LIN {X 0,Y 467.584,Z 526.238,A -85,B 0,C 180,E1 -7502.759,E2 -7502.759} C_VEL
LIN {X 0,Y 467.555,Z 526.241,A -85,B 0,C 180,E1 -7505.891,E2 -7505.891} C_VEL
LIN {X 0,Y 467.584,Z 526.242,A -85,B 0,C 180,E1 -7509.146,E2 -7509.146} C_VEL
LIN {X 0,Y 467.589,Z 526.235,A -85,B 0,C 180,E1 -7512.568,E2 -7512.568} C_VEL
LIN {X 0,Y 467.573,Z 526.241,A -85,B 0,C 180,E1 -7515.054,E2 -7515.054} C_VEL
LIN {X 0,Y 467.592,Z 526.243,A -85,B 0,C 180,E1 -7517.441,E2 -7517.441} C_VEL
LIN {X 0,Y 467.585,Z 526.237,A -85,B 0,C 180,E1 -7520.856,E2 -7520.856} C_VEL
LIN {X 0,Y 467.563,Z 526.239,A -85,B 0,C 180,E1 -7524.262,E2 -7524.262} C_VEL
LIN {X 0,Y 467.586,Z 526.241,A -85,B 0,C 180,E1 -7527.322,E2 -7527.322} C_VEL
LIN {X 0,Y 467.574,Z 526.237,A -85,B 0,C 180,E1 -7530.668,E2 -7530.668} C_VEL
LIN {X 0,Y 467.62,Z 526.235,A -85,B 0,C 180,E1 -7533.201,E2 -7533.201} C_VEL
LIN {X 0,Y 467.598,Z 526.234,A -85,B 0,C 180,E1 -7536.469,E2 -7536.469} C_VEL
LIN {X 0,Y 467.628,Z 526.237,A -85,B 0,C 180,E1 -7539.778,E2 -7539.778} C_VEL
LIN {X 0,Y 467.604,Z 526.233,A -85,B 0,C 180,E1 -7542.507,E2 -7542.507} C_VEL
LIN {X 0,Y 467.612,Z 526.234,A -85,B 0,C 180,E1 -7545.197,E2 -7545.197} C_VEL
LIN {X 0,Y 467.662,Z 526.232,A -85,B 0,C 180,E1 -7547.855,E2 -7547.855} C_VEL
LIN {X 0,Y 467.686,Z 526.226,A -85,B 0,C 180,E1 -7551.358,E2 -7551.358} C_VEL
LIN {X 0,Y 467.744,Z 526.221,A -85,B 0,C 180,E1 -7553.963,E2 -7553.963} C_VEL
LIN {X 0,Y 467.865,Z 526.204,A -85,B 0,C 180,E1 -7557.418,E2 -7557.418} C_VEL
LIN {X 0,Y 467.889,Z 526.204,A -85,B 0,C 180,E1 -7560,E2 -7560} C_VEL
LIN {X 0,Y 467.866,Z 526.201,A -85,B 0,C 180,E1 -7562.583,E2 -7562.583} C_VEL
LIN {X 0,Y 467.75,Z 526.221,A -85,B 0,C 180,E1 -7566.038,E2 -7566.038} C_VEL
LIN {X 0,Y 467.687,Z 526.223,A -85,B 0,C 180,E1 -7568.643,E2 -7568.643} C_VEL
LIN {X 0,Y 467.662,Z 526.229,A -85,B 0,C 180,E1 -7572.358,E2 -7572.358} C_VEL
LIN {X 0,Y 467.657,Z 526.234,A -85,B 0,C 180,E1 -7575.885,E2 -7575.885} C_VEL
LIN {X 0,Y 467.63,Z 526.231,A -85,B 0,C 180,E1 -7579.308,E2 -7579.308} C_VEL
LIN {X 0,Y 467.542,Z 526.249,A -85,B 0,C 180,E1 -7582.074,E2 -7582.074} C_VEL
LIN {X 0,Y 467.593,Z 526.235,A -85,B 0,C 180,E1 -7584.888,E2 -7584.888} C_VEL
LIN {X 0,Y 467.628,Z 526.234,A -85,B 0,C 180,E1 -7587.769,E2 -7587.769} C_VEL
LIN {X 0,Y 467.575,Z 526.237,A -85,B 0,C 180,E1 -7591.045,E2 -7591.045} C_VEL
LIN {X 0,Y 467.596,Z 526.242,A -85,B 0,C 180,E1 -7594.242,E2 -7594.242} C_VEL
LIN {X 0,Y 467.557,Z 526.239,A -85,B 0,C 180,E1 -7597.186,E2 -7597.186} C_VEL
LIN {X 0,Y 467.579,Z 526.245,A -85,B 0,C 180,E1 -7600.265,E2 -7600.265} C_VEL
LIN {X 0,Y 467.555,Z 526.241,A -85,B 0,C 180,E1 -7603.745,E2 -7603.745} C_VEL
LIN {X 0,Y 467.561,Z 526.247,A -85,B 0,C 180,E1 -7606.255,E2 -7606.255} C_VEL
LIN {X 0,Y 467.585,Z 526.239,A -85,B 0,C 180,E1 -7608.723,E2 -7608.723} C_VEL
LIN {X 0,Y 467.572,Z 526.24,A -85,B 0,C 180,E1 -7611.955,E2 -7611.955} C_VEL
LIN {X 0,Y 467.571,Z 526.238,A -85,B 0,C 180,E1 -7615.167,E2 -7615.167} C_VEL
LIN {X 0,Y 467.59,Z 526.241,A -85,B 0,C 180,E1 -7618.259,E2 -7618.259} C_VEL
LIN {X 0,Y 467.583,Z 526.238,A -85,B 0,C 180,E1 -7621.25,E2 -7621.25} C_VEL
LIN {X 0,Y 467.642,Z 526.251,A -85,B 0,C 180,E1 -7624.2,E2 -7624.2} C_VEL
LIN {X 0,Y 469.788,Z 537.488,A -85,B 0,C 180,E1 -7626.41,E2 -7626.41} C_VEL
LIN {X 0,Y 469.685,Z 545.066,A -85,B 0,C 180,E1 -7627.8,E2 -7627.8} C_VEL
LIN {X 0,Y 468.864,Z 562.445,A -85,B 0,C 180,E1 -7630.92,E2 -7630.92} C_VEL
LIN {X 0,Y 468.38,Z 574.086,A -85,B 0,C 180,E1 -7632.985,E2 -7632.985} C_VEL
LIN {X 0,Y 471.256,Z 592.032,A -85,B 0,C 180,E1 -7633.385,E2 -7633.385} C_VEL
LIN {X 0,Y 470.5,Z 682.57,A -85,B 0,C 180,E1 -7634.818,E2 -7634.818} C_VEL
LIN {X 0,Y 470.126,Z 695.682,A -85,B 0,C 180,E1 -7635.193,E2 -7635.193} C_VEL
LIN {X 0,Y 469.694,Z 707.78,A -85,B 0,C 180,E1 -7635.705,E2 -7635.705} C_VEL
LIN {X 0,Y 469.237,Z 719.207,A -85,B 0,C 180,E1 -7636.354,E2 -7636.354} C_VEL
LIN {X 0,Y 468.71,Z 731,A -85,B 0,C 180,E1 -7637.225,E2 -7637.225} C_VEL
LIN {X 0,Y 468.271,Z 741.513,A -85,B 0,C 180,E1 -7638.199,E2 -7638.199} C_VEL
LIN {X 0,Y 467.801,Z 750.137,A -85,B 0,C 180,E1 -7639.175,E2 -7639.175} C_VEL
LIN {X 0,Y 467.472,Z 758.092,A -85,B 0,C 180,E1 -7640.261,E2 -7640.261} C_VEL
LIN {X 0,Y 467.129,Z 765.864,A -85,B 0,C 180,E1 -7641.564,E2 -7641.564} C_VEL
LIN {X 0,Y 466.861,Z 773.006,A -85,B 0,C 180,E1 -7643.082,E2 -7643.082} C_VEL
LIN {X 0,Y 466.784,Z 777.763,A -85,B 0,C 180,E1 -7644.383,E2 -7644.383} C_VEL
LIN {X 0,Y 466.653,Z 781.394,A -85,B 0,C 180,E1 -7645.68,E2 -7645.68} C_VEL
LIN {X 0,Y 466.691,Z 783.27,A -85,B 0,C 180,E1 -7646.545,E2 -7646.545} C_VEL
LIN {X 0,Y 466.662,Z 784.674,A -85,B 0,C 180,E1 -7647.409,E2 -7647.409} C_VEL
LIN {X 0,Y 466.619,Z 786.281,A -85,B 0,C 180,E1 -7649.136,E2 -7649.136} C_VEL
LIN {X 0,Y 466.598,Z 786.495,A -85,B 0,C 180,E1 -7649.999,E2 -7649.999} C_VEL
LIN {X 0,Y 466.618,Z 786.274,A -85,B 0,C 180,E1 -7650.862,E2 -7650.862} C_VEL
LIN {X 0,Y 466.662,Z 784.653,A -85,B 0,C 180,E1 -7652.588,E2 -7652.588} C_VEL
LIN {X 0,Y 466.691,Z 783.242,A -85,B 0,C 180,E1 -7653.452,E2 -7653.452} C_VEL
LIN {X 0,Y 466.695,Z 780.279,A -85,B 0,C 180,E1 -7654.75,E2 -7654.75} C_VEL
LIN {X 0,Y 466.776,Z 776.271,A -85,B 0,C 180,E1 -7656.049,E2 -7656.049} C_VEL
LIN {X 0,Y 466.951,Z 770.103,A -85,B 0,C 180,E1 -7657.566,E2 -7657.566} C_VEL
LIN {X 0,Y 467.235,Z 763.371,A -85,B 0,C 180,E1 -7658.868,E2 -7658.868} C_VEL
LIN {X 0,Y 467.58,Z 755.016,A -85,B 0,C 180,E1 -7660.171,E2 -7660.171} C_VEL
LIN {X 0,Y 468.025,Z 746.436,A -85,B 0,C 180,E1 -7661.256,E2 -7661.256} C_VEL
LIN {X 0,Y 468.539,Z 736.228,A -85,B 0,C 180,E1 -7662.305,E2 -7662.305} C_VEL
LIN {X 0,Y 469.004,Z 725.64,A -85,B 0,C 180,E1 -7663.186,E2 -7663.186} C_VEL
LIN {X 0,Y 469.445,Z 713.811,A -85,B 0,C 180,E1 -7663.968,E2 -7663.968} C_VEL
LIN {X 0,Y 469.934,Z 701.861,A -85,B 0,C 180,E1 -7664.561,E2 -7664.561} C_VEL
LIN {X 0,Y 470.29,Z 688.979,A -85,B 0,C 180,E1 -7665.02,E2 -7665.02} C_VEL
LIN {X 0,Y 470.579,Z 675.477,A -85,B 0,C 180,E1 -7665.316,E2 -7665.316} C_VEL
LIN {X 0,Y 471.131,Z 591.332,A -85,B 0,C 180,E1 -7666.634,E2 -7666.634} C_VEL
LIN {X 0,Y 468.368,Z 573.742,A -85,B 0,C 180,E1 -7667.03,E2 -7667.03} C_VEL
LIN {X 0,Y 468.993,Z 557.448,A -85,B 0,C 180,E1 -7669.931,E2 -7669.931} C_VEL
LIN {X 0,Y 469.844,Z 541.073,A -85,B 0,C 180,E1 -7672.885,E2 -7672.885} C_VEL
LIN {X 0,Y 469.768,Z 537.298,A -85,B 0,C 180,E1 -7673.589,E2 -7673.589} C_VEL
LIN {X 0,Y 467.64,Z 526.237,A -85,B 0,C 180,E1 -7675.797,E2 -7675.797} C_VEL
LIN {X 0,Y 467.575,Z 526.245,A -85,B 0,C 180,E1 -7678.748,E2 -7678.748} C_VEL
LIN {X 0,Y 467.581,Z 526.244,A -85,B 0,C 180,E1 -7681.738,E2 -7681.738} C_VEL
LIN {X 0,Y 467.563,Z 526.241,A -85,B 0,C 180,E1 -7684.831,E2 -7684.831} C_VEL
LIN {X 0,Y 467.567,Z 526.243,A -85,B 0,C 180,E1 -7688.042,E2 -7688.042} C_VEL
LIN {X 0,Y 467.591,Z 526.239,A -85,B 0,C 180,E1 -7690.261,E2 -7690.261} C_VEL
LIN {X 0,Y 467.581,Z 526.24,A -85,B 0,C 180,E1 -7692.566,E2 -7692.566} C_VEL
LIN {X 0,Y 467.564,Z 526.245,A -85,B 0,C 180,E1 -7695.052,E2 -7695.052} C_VEL
LIN {X 0,Y 467.582,Z 526.243,A -85,B 0,C 180,E1 -7697.439,E2 -7697.439} C_VEL
LIN {X 0,Y 467.608,Z 526.235,A -85,B 0,C 180,E1 -7700.857,E2 -7700.857} C_VEL
LIN {X 0,Y 467.556,Z 526.241,A -85,B 0,C 180,E1 -7704.259,E2 -7704.259} C_VEL
LIN {X 0,Y 467.574,Z 526.243,A -85,B 0,C 180,E1 -7707.32,E2 -7707.32} C_VEL
LIN {X 0,Y 467.569,Z 526.239,A -85,B 0,C 180,E1 -7710.664,E2 -7710.664} C_VEL
LIN {X 0,Y 467.619,Z 526.234,A -85,B 0,C 180,E1 -7713.199,E2 -7713.199} C_VEL
LIN {X 0,Y 467.583,Z 526.233,A -85,B 0,C 180,E1 -7716.467,E2 -7716.467} C_VEL
LIN {X 0,Y 467.614,Z 526.232,A -85,B 0,C 180,E1 -7719.776,E2 -7719.776} C_VEL
LIN {X 0,Y 467.599,Z 526.235,A -85,B 0,C 180,E1 -7722.506,E2 -7722.506} C_VEL
LIN {X 0,Y 467.599,Z 526.236,A -85,B 0,C 180,E1 -7725.196,E2 -7725.196} C_VEL
LIN {X 0,Y 467.672,Z 526.226,A -85,B 0,C 180,E1 -7727.855,E2 -7727.855} C_VEL
LIN {X 0,Y 467.672,Z 526.23,A -85,B 0,C 180,E1 -7731.357,E2 -7731.357} C_VEL
LIN {X 0,Y 467.733,Z 526.22,A -85,B 0,C 180,E1 -7733.962,E2 -7733.962} C_VEL
LIN {X 0,Y 467.85,Z 526.211,A -85,B 0,C 180,E1 -7737.417,E2 -7737.417} C_VEL
LIN {X 0,Y 467.871,Z 526.203,A -85,B 0,C 180,E1 -7740,E2 -7740} C_VEL
LIN {X 0,Y 467.85,Z 526.203,A -85,B 0,C 180,E1 -7742.583,E2 -7742.583} C_VEL
LIN {X 0,Y 467.741,Z 526.219,A -85,B 0,C 180,E1 -7746.037,E2 -7746.037} C_VEL
LIN {X 0,Y 467.671,Z 526.227,A -85,B 0,C 180,E1 -7748.642,E2 -7748.642} C_VEL
LIN {X 0,Y 467.678,Z 526.226,A -85,B 0,C 180,E1 -7752.379,E2 -7752.379} C_VEL
LIN {X 0,Y 467.637,Z 526.235,A -85,B 0,C 180,E1 -7755.885,E2 -7755.885} C_VEL
LIN {X 0,Y 467.612,Z 526.241,A -85,B 0,C 180,E1 -7759.308,E2 -7759.308} C_VEL
LIN {X 0,Y 467.523,Z 526.248,A -85,B 0,C 180,E1 -7762.074,E2 -7762.074} C_VEL
LIN {X 0,Y 467.591,Z 526.241,A -85,B 0,C 180,E1 -7764.887,E2 -7764.887} C_VEL
LIN {X 0,Y 467.628,Z 526.269,A -85,B 0,C 180,E1 -7767.951,E2 -7767.951} C_VEL
LIN {X 0,Y 469.093,Z 534.649,A -85,B 0,C 180,E1 -7769.877,E2 -7769.877} C_VEL
LIN {X 0,Y 468.524,Z 548.568,A -85,B 0,C 180,E1 -7772.861,E2 -7772.861} C_VEL
LIN {X 0,Y 468.485,Z 549.397,A -85,B 0,C 180,E1 -7773.037,E2 -7773.037} C_VEL
LIN {X 0,Y 471.331,Z 564.269,A -85,B 0,C 180,E1 -7773.396,E2 -7773.396} C_VEL
LIN {X 0,Y 470.507,Z 656.723,A -85,B 0,C 180,E1 -7774.868,E2 -7774.868} C_VEL
LIN {X 0,Y 470.226,Z 670.141,A -85,B 0,C 180,E1 -7775.263,E2 -7775.263} C_VEL
LIN {X 0,Y 469.853,Z 681.913,A -85,B 0,C 180,E1 -7775.771,E2 -7775.771} C_VEL
LIN {X 0,Y 469.439,Z 692.978,A -85,B 0,C 180,E1 -7776.407,E2 -7776.407} C_VEL
LIN {X 0,Y 468.925,Z 704.749,A -85,B 0,C 180,E1 -7777.283,E2 -7777.283} C_VEL
LIN {X 0,Y 468.474,Z 714.85,A -85,B 0,C 180,E1 -7778.224,E2 -7778.224} C_VEL
LIN {X 0,Y 468.041,Z 723.751,A -85,B 0,C 180,E1 -7779.237,E2 -7779.237} C_VEL
LIN {X 0,Y 467.686,Z 731.139,A -85,B 0,C 180,E1 -7780.253,E2 -7780.253} C_VEL
LIN {X 0,Y 467.345,Z 738.241,A -85,B 0,C 180,E1 -7781.427,E2 -7781.427} C_VEL
LIN {X 0,Y 467.031,Z 745.32,A -85,B 0,C 180,E1 -7782.897,E2 -7782.897} C_VEL
LIN {X 0,Y 466.844,Z 750.861,A -85,B 0,C 180,E1 -7784.392,E2 -7784.392} C_VEL
LIN {X 0,Y 466.665,Z 754.261,A -85,B 0,C 180,E1 -7785.6,E2 -7785.6} C_VEL
LIN {X 0,Y 466.645,Z 755.815,A -85,B 0,C 180,E1 -7786.295,E2 -7786.295} C_VEL
LIN {X 0,Y 466.541,Z 757.954,A -85,B 0,C 180,E1 -7787.572,E2 -7787.572} C_VEL
LIN {X 0,Y 466.473,Z 759.216,A -85,B 0,C 180,E1 -7788.877,E2 -7788.877} C_VEL
LIN {X 0,Y 466.495,Z 759.567,A -85,B 0,C 180,E1 -7790.204,E2 -7790.204} C_VEL
LIN {X 0,Y 466.545,Z 758.676,A -85,B 0,C 180,E1 -7791.859,E2 -7791.859} C_VEL
LIN {X 0,Y 466.613,Z 756.359,A -85,B 0,C 180,E1 -7793.503,E2 -7793.503} C_VEL
LIN {X 0,Y 466.747,Z 752.589,A -85,B 0,C 180,E1 -7795.099,E2 -7795.099} C_VEL
LIN {X 0,Y 466.765,Z 751.849,A -85,B 0,C 180,E1 -7795.354,E2 -7795.354} C_VEL
LIN {X 0,Y 466.167,Z 749.789,A -85,B 0,C 180,E1 -7796.032,E2 -7796.032} C_VEL
LIN {X 0,Y 463.443,Z 746.027,A -85,B 0,C 180,E1 -7797.115,E2 -7797.115} C_VEL
LIN {X 0,Y 460.774,Z 741.545,A -85,B 0,C 180,E1 -7798.164,E2 -7798.164} C_VEL
LIN {X 0,Y 460.265,Z 738.355,A -85,B 0,C 180,E1 -7798.782,E2 -7798.782} C_VEL
LIN {X 0,Y 460.686,Z 730.288,A -85,B 0,C 180,E1 -7800.115,E2 -7800.115} C_VEL
LIN {X 0,Y 461.126,Z 721.369,A -85,B 0,C 180,E1 -7801.31,E2 -7801.31} C_VEL
LIN {X 0,Y 461.626,Z 711.879,A -85,B 0,C 180,E1 -7802.346,E2 -7802.346} C_VEL
LIN {X 0,Y 462.226,Z 700.526,A -85,B 0,C 180,E1 -7803.333,E2 -7803.333} C_VEL
LIN {X 0,Y 462.71,Z 688.324,A -85,B 0,C 180,E1 -7804.17,E2 -7804.17} C_VEL
LIN {X 0,Y 463.133,Z 676.128,A -85,B 0,C 180,E1 -7804.797,E2 -7804.797} C_VEL
LIN {X 0,Y 463.552,Z 663.091,A -85,B 0,C 180,E1 -7805.271,E2 -7805.271} C_VEL
LIN {X 0,Y 463.735,Z 651.259,A -85,B 0,C 180,E1 -7805.546,E2 -7805.546} C_VEL
LIN {X 0,Y 464.458,Z 564.756,A -85,B 0,C 180,E1 -7806.922,E2 -7806.922} C_VEL
LIN {X 0,Y 461.484,Z 549.204,A -85,B 0,C 180,E1 -7807.298,E2 -7807.298} C_VEL
LIN {X 0,Y 462.003,Z 535.66,A -85,B 0,C 180,E1 -7810.218,E2 -7810.218} C_VEL
LIN {X 0,Y 460.604,Z 527.111,A -85,B 0,C 180,E1 -7812.176,E2 -7812.176} C_VEL
LIN {X 0,Y 460.561,Z 527.119,A -85,B 0,C 180,E1 -7814.966,E2 -7814.966} C_VEL
LIN {X 0,Y 460.604,Z 527.105,A -85,B 0,C 180,E1 -7817.667,E2 -7817.667} C_VEL
LIN {X 0,Y 460.624,Z 527.106,A -85,B 0,C 180,E1 -7821.225,E2 -7821.225} C_VEL
LIN {X 0,Y 460.698,Z 527.093,A -85,B 0,C 180,E1 -7823.871,E2 -7823.871} C_VEL
LIN {X 0,Y 460.823,Z 527.08,A -85,B 0,C 180,E1 -7827.379,E2 -7827.379} C_VEL
LIN {X 0,Y 460.851,Z 527.074,A -85,B 0,C 180,E1 -7830.001,E2 -7830.001} C_VEL
LIN {X 0,Y 460.822,Z 527.082,A -85,B 0,C 180,E1 -7832.624,E2 -7832.624} C_VEL
LIN {X 0,Y 460.699,Z 527.093,A -85,B 0,C 180,E1 -7836.131,E2 -7836.131} C_VEL
LIN {X 0,Y 460.627,Z 527.107,A -85,B 0,C 180,E1 -7838.777,E2 -7838.777} C_VEL
LIN {X 0,Y 460.612,Z 527.105,A -85,B 0,C 180,E1 -7842.446,E2 -7842.446} C_VEL
LIN {X 0,Y 460.599,Z 527.106,A -85,B 0,C 180,E1 -7845.999,E2 -7845.999} C_VEL
LIN {X 0,Y 460.568,Z 527.112,A -85,B 0,C 180,E1 -7849.617,E2 -7849.617} C_VEL
LIN {X 0,Y 460.51,Z 527.117,A -85,B 0,C 180,E1 -7852.43,E2 -7852.43} C_VEL
LIN {X 0,Y 460.568,Z 527.111,A -85,B 0,C 180,E1 -7855.803,E2 -7855.803} C_VEL
LIN {X 0,Y 460.553,Z 527.111,A -85,B 0,C 180,E1 -7858.234,E2 -7858.234} C_VEL
LIN {X 0,Y 460.522,Z 527.123,A -85,B 0,C 180,E1 -7861.284,E2 -7861.284} C_VEL
LIN {X 0,Y 460.533,Z 527.114,A -85,B 0,C 180,E1 -7864.506,E2 -7864.506} C_VEL
LIN {X 0,Y 460.503,Z 527.122,A -85,B 0,C 180,E1 -7867.624,E2 -7867.624} C_VEL
LIN {X 0,Y 460.545,Z 527.112,A -85,B 0,C 180,E1 -7870.271,E2 -7870.271} C_VEL
LIN {X 0,Y 460.512,Z 527.125,A -85,B 0,C 180,E1 -7873.375,E2 -7873.375} C_VEL
LIN {X 0,Y 460.502,Z 527.118,A -85,B 0,C 180,E1 -7876.626,E2 -7876.626} C_VEL
LIN {X 0,Y 460.545,Z 527.117,A -85,B 0,C 180,E1 -7879.732,E2 -7879.732} C_VEL
LIN {X 0,Y 460.503,Z 527.118,A -85,B 0,C 180,E1 -7882.525,E2 -7882.525} C_VEL
LIN {X 0,Y 460.55,Z 527.118,A -85,B 0,C 180,E1 -7885.625,E2 -7885.625} C_VEL
LIN {X 0,Y 460.541,Z 527.113,A -85,B 0,C 180,E1 -7888.745,E2 -7888.745} C_VEL
LIN {X 0,Y 460.586,Z 527.108,A -85,B 0,C 180,E1 -7892.255,E2 -7892.255} C_VEL
LIN {X 0,Y 460.552,Z 527.112,A -85,B 0,C 180,E1 -7894.706,E2 -7894.706} C_VEL
LIN {X 0,Y 460.516,Z 527.124,A -85,B 0,C 180,E1 -7897.572,E2 -7897.572} C_VEL
LIN {X 0,Y 460.573,Z 527.109,A -85,B 0,C 180,E1 -7900.385,E2 -7900.385} C_VEL
LIN {X 0,Y 460.606,Z 527.109,A -85,B 0,C 180,E1 -7904.003,E2 -7904.003} C_VEL
LIN {X 0,Y 460.615,Z 527.112,A -85,B 0,C 180,E1 -7907.666,E2 -7907.666} C_VEL
LIN {X 0,Y 460.633,Z 527.104,A -85,B 0,C 180,E1 -7911.224,E2 -7911.224} C_VEL
LIN {X 0,Y 460.71,Z 527.099,A -85,B 0,C 180,E1 -7913.871,E2 -7913.871} C_VEL
LIN {X 0,Y 460.806,Z 527.083,A -85,B 0,C 180,E1 -7917.378,E2 -7917.378} C_VEL
LIN {X 0,Y 460.859,Z 527.079,A -85,B 0,C 180,E1 -7920,E2 -7920} C_VEL
LIN {X 0,Y 460.806,Z 527.08,A -85,B 0,C 180,E1 -7922.623,E2 -7922.623} C_VEL
LIN {X 0,Y 460.717,Z 527.096,A -85,B 0,C 180,E1 -7926.13,E2 -7926.13} C_VEL
LIN {X 0,Y 460.634,Z 527.101,A -85,B 0,C 180,E1 -7928.776,E2 -7928.776} C_VEL
LIN {X 0,Y 460.621,Z 527.105,A -85,B 0,C 180,E1 -7932.445,E2 -7932.445} C_VEL
LIN {X 0,Y 460.608,Z 527.113,A -85,B 0,C 180,E1 -7935.998,E2 -7935.998} C_VEL
LIN {X 0,Y 460.576,Z 527.112,A -85,B 0,C 180,E1 -7939.616,E2 -7939.616} C_VEL
LIN {X 0,Y 460.518,Z 527.119,A -85,B 0,C 180,E1 -7942.429,E2 -7942.429} C_VEL
LIN {X 0,Y 460.561,Z 527.115,A -85,B 0,C 180,E1 -7945.798,E2 -7945.798} C_VEL
LIN {X 0,Y 460.56,Z 527.117,A -85,B 0,C 180,E1 -7948.233,E2 -7948.233} C_VEL
LIN {X 0,Y 460.528,Z 527.115,A -85,B 0,C 180,E1 -7951.283,E2 -7951.283} C_VEL
LIN {X 0,Y 460.54,Z 527.117,A -85,B 0,C 180,E1 -7954.505,E2 -7954.505} C_VEL
LIN {X 0,Y 460.509,Z 527.118,A -85,B 0,C 180,E1 -7957.623,E2 -7957.623} C_VEL
LIN {X 0,Y 460.543,Z 527.121,A -85,B 0,C 180,E1 -7960.268,E2 -7960.268} C_VEL
LIN {X 0,Y 460.515,Z 527.116,A -85,B 0,C 180,E1 -7963.374,E2 -7963.374} C_VEL
LIN {X 0,Y 460.506,Z 527.121,A -85,B 0,C 180,E1 -7966.624,E2 -7966.624} C_VEL
LIN {X 0,Y 460.549,Z 527.113,A -85,B 0,C 180,E1 -7969.73,E2 -7969.73} C_VEL
LIN {X 0,Y 460.507,Z 527.123,A -85,B 0,C 180,E1 -7972.523,E2 -7972.523} C_VEL
LIN {X 0,Y 460.553,Z 527.112,A -85,B 0,C 180,E1 -7975.623,E2 -7975.623} C_VEL
LIN {X 0,Y 460.544,Z 527.119,A -85,B 0,C 180,E1 -7978.744,E2 -7978.744} C_VEL
LIN {X 0,Y 460.588,Z 527.115,A -85,B 0,C 180,E1 -7982.253,E2 -7982.253} C_VEL
LIN {X 0,Y 460.639,Z 527.249,A -85,B 0,C 180,E1 -7984.009,E2 -7984.009} C_VEL
LIN {X 0,Y 462.957,Z 539.818,A -85,B 0,C 180,E1 -7986.515,E2 -7986.515} C_VEL
LIN {X 0,Y 462.308,Z 553.699,A -85,B 0,C 180,E1 -7989.068,E2 -7989.068} C_VEL
LIN {X 0,Y 461.536,Z 571.352,A -85,B 0,C 180,E1 -7992.268,E2 -7992.268} C_VEL
LIN {X 0,Y 461.423,Z 573.949,A -85,B 0,C 180,E1 -7992.734,E2 -7992.734} C_VEL
LIN {X 0,Y 464.425,Z 593.483,A -85,B 0,C 180,E1 -7993.165,E2 -7993.165} C_VEL
LIN {X 0,Y 463.643,Z 682.087,A -85,B 0,C 180,E1 -7994.588,E2 -7994.588} C_VEL
LIN {X 0,Y 463.232,Z 695.286,A -85,B 0,C 180,E1 -7994.968,E2 -7994.968} C_VEL
LIN {X 0,Y 462.745,Z 708.554,A -85,B 0,C 180,E1 -7995.542,E2 -7995.542} C_VEL
LIN {X 0,Y 462.222,Z 720.503,A -85,B 0,C 180,E1 -7996.255,E2 -7996.255} C_VEL
LIN {X 0,Y 461.726,Z 731.59,A -85,B 0,C 180,E1 -7997.104,E2 -7997.104} C_VEL
LIN {X 0,Y 461.242,Z 742.316,A -85,B 0,C 180,E1 -7998.128,E2 -7998.128} C_VEL
LIN {X 0,Y 460.734,Z 751.598,A -85,B 0,C 180,E1 -7999.229,E2 -7999.229} C_VEL
LIN {X 0,Y 460.291,Z 760.617,A -85,B 0,C 180,E1 -8000.552,E2 -8000.552} C_VEL
LIN {X 0,Y 460.008,Z 767.882,A -85,B 0,C 180,E1 -8001.874,E2 -8001.874} C_VEL
LIN {X 0,Y 459.75,Z 773.966,A -85,B 0,C 180,E1 -8003.272,E2 -8003.272} C_VEL
LIN {X 0,Y 459.662,Z 778.871,A -85,B 0,C 180,E1 -8004.735,E2 -8004.735} C_VEL
LIN {X 0,Y 459.57,Z 781.18,A -85,B 0,C 180,E1 -8005.614,E2 -8005.614} C_VEL
LIN {X 0,Y 459.587,Z 783.059,A -85,B 0,C 180,E1 -8006.492,E2 -8006.492} C_VEL
LIN {X 0,Y 459.585,Z 784.466,A -85,B 0,C 180,E1 -8007.369,E2 -8007.369} C_VEL
LIN {X 0,Y 459.522,Z 786.075,A -85,B 0,C 180,E1 -8009.122,E2 -8009.122} C_VEL
LIN {X 0,Y 459.53,Z 786.291,A -85,B 0,C 180,E1 -8009.999,E2 -8009.999} C_VEL
LIN {X 0,Y 459.522,Z 786.07,A -85,B 0,C 180,E1 -8010.875,E2 -8010.875} C_VEL
LIN {X 0,Y 459.584,Z 784.448,A -85,B 0,C 180,E1 -8012.628,E2 -8012.628} C_VEL
LIN {X 0,Y 459.586,Z 783.035,A -85,B 0,C 180,E1 -8013.506,E2 -8013.506} C_VEL
LIN {X 0,Y 459.623,Z 780.07,A -85,B 0,C 180,E1 -8014.823,E2 -8014.823} C_VEL
LIN {X 0,Y 459.713,Z 775.019,A -85,B 0,C 180,E1 -8016.429,E2 -8016.429} C_VEL
LIN {X 0,Y 459.934,Z 768.867,A -85,B 0,C 180,E1 -8017.903,E2 -8017.903} C_VEL
LIN {X 0,Y 460.232,Z 761.9,A -85,B 0,C 180,E1 -8019.225,E2 -8019.225} C_VEL
LIN {X 0,Y 460.611,Z 753.172,A -85,B 0,C 180,E1 -8020.549,E2 -8020.549} C_VEL
LIN {X 0,Y 461.118,Z 744.231,A -85,B 0,C 180,E1 -8021.649,E2 -8021.649} C_VEL
LIN {X 0,Y 461.596,Z 734.395,A -85,B 0,C 180,E1 -8022.642,E2 -8022.642} C_VEL
LIN {X 0,Y 462.124,Z 723.639,A -85,B 0,C 180,E1 -8023.521,E2 -8023.521} C_VEL
LIN {X 0,Y 462.635,Z 711.554,A -85,B 0,C 180,E1 -8024.29,E2 -8024.29} C_VEL
LIN {X 0,Y 463.135,Z 698.986,A -85,B 0,C 180,E1 -8024.892,E2 -8024.892} C_VEL
LIN {X 0,Y 463.515,Z 686.861,A -85,B 0,C 180,E1 -8025.301,E2 -8025.301} C_VEL
LIN {X 0,Y 463.787,Z 671.695,A -85,B 0,C 180,E1 -8025.602,E2 -8025.602} C_VEL
LIN {X 0,Y 464.316,Z 591.83,A -85,B 0,C 180,E1 -8026.88,E2 -8026.88} C_VEL
LIN {X 0,Y 461.392,Z 573.556,A -85,B 0,C 180,E1 -8027.296,E2 -8027.296} C_VEL
LIN {X 0,Y 462.094,Z 557.28,A -85,B 0,C 180,E1 -8030.242,E2 -8030.242} C_VEL
LIN {X 0,Y 462.944,Z 540.944,A -85,B 0,C 180,E1 -8033.246,E2 -8033.246} C_VEL
LIN {X 0,Y 462.331,Z 535.913,A -85,B 0,C 180,E1 -8034.23,E2 -8034.23} C_VEL
LIN {X 0,Y 460.587,Z 527.115,A -85,B 0,C 180,E1 -8036.06,E2 -8036.06} C_VEL
LIN {X 0,Y 460.553,Z 527.12,A -85,B 0,C 180,E1 -8038.231,E2 -8038.231} C_VEL
LIN {X 0,Y 460.519,Z 527.124,A -85,B 0,C 180,E1 -8041.282,E2 -8041.282} C_VEL
LIN {X 0,Y 460.529,Z 527.117,A -85,B 0,C 180,E1 -8044.504,E2 -8044.504} C_VEL
LIN {X 0,Y 460.526,Z 527.125,A -85,B 0,C 180,E1 -8047.619,E2 -8047.619} C_VEL
LIN {X 0,Y 460.554,Z 527.116,A -85,B 0,C 180,E1 -8050.271,E2 -8050.271} C_VEL
LIN {X 0,Y 460.503,Z 527.128,A -85,B 0,C 180,E1 -8053.373,E2 -8053.373} C_VEL
LIN {X 0,Y 460.493,Z 527.122,A -85,B 0,C 180,E1 -8056.623,E2 -8056.623} C_VEL
LIN {X 0,Y 460.551,Z 527.117,A -85,B 0,C 180,E1 -8059.727,E2 -8059.727} C_VEL
LIN {X 0,Y 460.521,Z 527.115,A -85,B 0,C 180,E1 -8062.518,E2 -8062.518} C_VEL
LIN {X 0,Y 460.541,Z 527.117,A -85,B 0,C 180,E1 -8065.623,E2 -8065.623} C_VEL
LIN {X 0,Y 460.528,Z 527.116,A -85,B 0,C 180,E1 -8068.743,E2 -8068.743} C_VEL
LIN {X 0,Y 460.55,Z 527.115,A -85,B 0,C 180,E1 -8071.766,E2 -8071.766} C_VEL
LIN {X 0,Y 460.55,Z 527.114,A -85,B 0,C 180,E1 -8074.704,E2 -8074.704} C_VEL
LIN {X 0,Y 460.502,Z 527.125,A -85,B 0,C 180,E1 -8077.57,E2 -8077.57} C_VEL
LIN {X 0,Y 460.559,Z 527.107,A -85,B 0,C 180,E1 -8080.384,E2 -8080.384} C_VEL
LIN {X 0,Y 460.555,Z 527.117,A -85,B 0,C 180,E1 -8083.145,E2 -8083.145} C_VEL
LIN {X 0,Y 460.547,Z 527.116,A -85,B 0,C 180,E1 -8085.867,E2 -8085.867} C_VEL
LIN {X 0,Y 460.621,Z 527.101,A -85,B 0,C 180,E1 -8088.559,E2 -8088.559} C_VEL
LIN {X 0,Y 460.684,Z 527.095,A -85,B 0,C 180,E1 -8092.108,E2 -8092.108} C_VEL
LIN {X 0,Y 460.688,Z 527.096,A -85,B 0,C 180,E1 -8094.748,E2 -8094.748} C_VEL
LIN {X 0,Y 460.815,Z 527.088,A -85,B 0,C 180,E1 -8097.377,E2 -8097.377} C_VEL
LIN {X 0,Y 460.842,Z 527.079,A -85,B 0,C 180,E1 -8100,E2 -8100} C_VEL
LIN {X 0,Y 460.815,Z 527.08,A -85,B 0,C 180,E1 -8102.622,E2 -8102.622} C_VEL
LIN {X 0,Y 460.705,Z 527.095,A -85,B 0,C 180,E1 -8106.13,E2 -8106.13} C_VEL
LIN {X 0,Y 460.618,Z 527.107,A -85,B 0,C 180,E1 -8108.776,E2 -8108.776} C_VEL
LIN {X 0,Y 460.621,Z 527.106,A -85,B 0,C 180,E1 -8112.457,E2 -8112.457} C_VEL
LIN {X 0,Y 460.587,Z 527.113,A -85,B 0,C 180,E1 -8115.998,E2 -8115.998} C_VEL
LIN {X 0,Y 460.558,Z 527.117,A -85,B 0,C 180,E1 -8118.902,E2 -8118.902} C_VEL
LIN {X 0,Y 460.503,Z 527.123,A -85,B 0,C 180,E1 -8121.486,E2 -8121.486} C_VEL
LIN {X 0,Y 460.53,Z 527.119,A -85,B 0,C 180,E1 -8124.332,E2 -8124.332} C_VEL
LIN {X 0,Y 460.598,Z 527.115,A -85,B 0,C 180,E1 -8127.727,E2 -8127.727} C_VEL
LIN {X 0,Y 462.016,Z 534.767,A -85,B 0,C 180,E1 -8129.525,E2 -8129.525} C_VEL
LIN {X 0,Y 461.907,Z 542.158,A -85,B 0,C 180,E1 -8131.152,E2 -8131.152} C_VEL
LIN {X 0,Y 461.546,Z 549.686,A -85,B 0,C 180,E1 -8132.777,E2 -8132.777} C_VEL
LIN {X 0,Y 464.587,Z 565.361,A -85,B 0,C 180,E1 -8133.156,E2 -8133.156} C_VEL
LIN {X 0,Y 463.681,Z 656.87,A -85,B 0,C 180,E1 -8134.637,E2 -8134.637} C_VEL
LIN {X 0,Y 463.412,Z 669.859,A -85,B 0,C 180,E1 -8135.023,E2 -8135.023} C_VEL
LIN {X 0,Y 462.989,Z 682.207,A -85,B 0,C 180,E1 -8135.56,E2 -8135.56} C_VEL
LIN {X 0,Y 462.515,Z 694.146,A -85,B 0,C 180,E1 -8136.268,E2 -8136.268} C_VEL
LIN {X 0,Y 462.011,Z 704.688,A -85,B 0,C 180,E1 -8137.067,E2 -8137.067} C_VEL
LIN {X 0,Y 461.503,Z 715.82,A -85,B 0,C 180,E1 -8138.125,E2 -8138.125} C_VEL
LIN {X 0,Y 461.03,Z 724.511,A -85,B 0,C 180,E1 -8139.142,E2 -8139.142} C_VEL
LIN {X 0,Y 460.568,Z 733.341,A -85,B 0,C 180,E1 -8140.417,E2 -8140.417} C_VEL
LIN {X 0,Y 460.15,Z 741.357,A -85,B 0,C 180,E1 -8141.863,E2 -8141.863} C_VEL
LIN {X 0,Y 459.947,Z 746.821,A -85,B 0,C 180,E1 -8143.104,E2 -8143.104} C_VEL
LIN {X 0,Y 459.716,Z 752.229,A -85,B 0,C 180,E1 -8144.686,E2 -8144.686} C_VEL
LIN {X 0,Y 459.561,Z 755.447,A -85,B 0,C 180,E1 -8145.952,E2 -8145.952} C_VEL
LIN {X 0,Y 459.489,Z 757.776,A -85,B 0,C 180,E1 -8147.236,E2 -8147.236} C_VEL
LIN {X 0,Y 459.389,Z 759.427,A -85,B 0,C 180,E1 -8148.867,E2 -8148.867} C_VEL
LIN {X 0,Y 459.413,Z 759.795,A -85,B 0,C 180,E1 -8150.023,E2 -8150.023} C_VEL
LIN {X 0,Y 459.397,Z 759.374,A -85,B 0,C 180,E1 -8151.279,E2 -8151.279} C_VEL
LIN {X 0,Y 459.458,Z 757.939,A -85,B 0,C 180,E1 -8152.693,E2 -8152.693} C_VEL
LIN {X 0,Y 459.62,Z 755.375,A -85,B 0,C 180,E1 -8154.136,E2 -8154.136} C_VEL
LIN {X 0,Y 459.727,Z 751.44,A -85,B 0,C 180,E1 -8155.64,E2 -8155.64} C_VEL
LIN {X 0,Y 459.969,Z 745.914,A -85,B 0,C 180,E1 -8157.177,E2 -8157.177} C_VEL
LIN {X 0,Y 460.251,Z 738.672,A -85,B 0,C 180,E1 -8158.725,E2 -8158.725} C_VEL
LIN {X 0,Y 460.265,Z 738.355,A -85,B 0,C 180,E1 -8158.782,E2 -8158.782} C_VEL
LIN {X 0,Y 459.779,Z 735.039,A -85,B 0,C 180,E1 -8159.384,E2 -8159.384} C_VEL
LIN {X 0,Y 457.246,Z 729.311,A -85,B 0,C 180,E1 -8160.35,E2 -8160.35} C_VEL
LIN {X 0,Y 454.746,Z 723.099,A -85,B 0,C 180,E1 -8161.271,E2 -8161.271} C_VEL
LIN {X 0,Y 454.312,Z 718.898,A -85,B 0,C 180,E1 -8161.793,E2 -8161.793} C_VEL
LIN {X 0,Y 454.824,Z 708.378,A -85,B 0,C 180,E1 -8162.883,E2 -8162.883} C_VEL
LIN {X 0,Y 455.428,Z 697.388,A -85,B 0,C 180,E1 -8163.787,E2 -8163.787} C_VEL
LIN {X 0,Y 455.938,Z 684.607,A -85,B 0,C 180,E1 -8164.603,E2 -8164.603} C_VEL
LIN {X 0,Y 456.414,Z 671.786,A -85,B 0,C 180,E1 -8165.207,E2 -8165.207} C_VEL
LIN {X 0,Y 456.722,Z 658.866,A -85,B 0,C 180,E1 -8165.619,E2 -8165.619} C_VEL
LIN {X 0,Y 456.98,Z 638.88,A -85,B 0,C 180,E1 -8165.981,E2 -8165.981} C_VEL
LIN {X 0,Y 457.704,Z 565.843,A -85,B 0,C 180,E1 -8167.159,E2 -8167.159} C_VEL
LIN {X 0,Y 454.539,Z 549.358,A -85,B 0,C 180,E1 -8167.572,E2 -8167.572} C_VEL
LIN {X 0,Y 455.078,Z 537.586,A -85,B 0,C 180,E1 -8170.139,E2 -8170.139} C_VEL
LIN {X 0,Y 453.686,Z 528.74,A -85,B 0,C 180,E1 -8172.186,E2 -8172.186} C_VEL
LIN {X 0,Y 453.535,Z 527.992,A -85,B 0,C 180,E1 -8172.413,E2 -8172.413} C_VEL
LIN {X 0,Y 453.535,Z 527.994,A -85,B 0,C 180,E1 -8174.728,E2 -8174.728} C_VEL
LIN {X 0,Y 453.558,Z 527.984,A -85,B 0,C 180,E1 -8177.472,E2 -8177.472} C_VEL
LIN {X 0,Y 453.588,Z 527.984,A -85,B 0,C 180,E1 -8181.088,E2 -8181.088} C_VEL
LIN {X 0,Y 453.666,Z 527.969,A -85,B 0,C 180,E1 -8183.776,E2 -8183.776} C_VEL
LIN {X 0,Y 453.763,Z 527.96,A -85,B 0,C 180,E1 -8187.338,E2 -8187.338} C_VEL
LIN {X 0,Y 453.821,Z 527.95,A -85,B 0,C 180,E1 -8190.001,E2 -8190.001} C_VEL
LIN {X 0,Y 453.763,Z 527.962,A -85,B 0,C 180,E1 -8192.664,E2 -8192.664} C_VEL
LIN {X 0,Y 453.667,Z 527.97,A -85,B 0,C 180,E1 -8196.227,E2 -8196.227} C_VEL
LIN {X 0,Y 453.59,Z 527.986,A -85,B 0,C 180,E1 -8198.915,E2 -8198.915} C_VEL
LIN {X 0,Y 453.562,Z 527.984,A -85,B 0,C 180,E1 -8202.53,E2 -8202.53} C_VEL
LIN {X 0,Y 453.543,Z 527.985,A -85,B 0,C 180,E1 -8206.197,E2 -8206.197} C_VEL
LIN {X 0,Y 453.517,Z 527.995,A -85,B 0,C 180,E1 -8209.041,E2 -8209.041} C_VEL
LIN {X 0,Y 453.476,Z 527.994,A -85,B 0,C 180,E1 -8211.837,E2 -8211.837} C_VEL
LIN {X 0,Y 453.513,Z 527.991,A -85,B 0,C 180,E1 -8214.736,E2 -8214.736} C_VEL
LIN {X 0,Y 453.533,Z 527.986,A -85,B 0,C 180,E1 -8217.961,E2 -8217.961} C_VEL
LIN {X 0,Y 453.467,Z 527.999,A -85,B 0,C 180,E1 -8221.526,E2 -8221.526} C_VEL
LIN {X 0,Y 453.488,Z 527.994,A -85,B 0,C 180,E1 -8224.778,E2 -8224.778} C_VEL
LIN {X 0,Y 453.466,Z 527.994,A -85,B 0,C 180,E1 -8228.313,E2 -8228.313} C_VEL
LIN {X 0,Y 453.497,Z 527.991,A -85,B 0,C 180,E1 -8230.61,E2 -8230.61} C_VEL
LIN {X 0,Y 453.466,Z 528.001,A -85,B 0,C 180,E1 -8233.246,E2 -8233.246} C_VEL
LIN {X 0,Y 453.469,Z 527.997,A -85,B 0,C 180,E1 -8235.78,E2 -8235.78} C_VEL
LIN {X 0,Y 453.482,Z 527.993,A -85,B 0,C 180,E1 -8238.21,E2 -8238.21} C_VEL
LIN {X 0,Y 453.498,Z 527.992,A -85,B 0,C 180,E1 -8240.794,E2 -8240.794} C_VEL
LIN {X 0,Y 453.458,Z 527.998,A -85,B 0,C 180,E1 -8243.918,E2 -8243.918} C_VEL
LIN {X 0,Y 453.487,Z 527.995,A -85,B 0,C 180,E1 -8247.152,E2 -8247.152} C_VEL
LIN {X 0,Y 453.479,Z 527.993,A -85,B 0,C 180,E1 -8250.269,E2 -8250.269} C_VEL
LIN {X 0,Y 453.509,Z 527.994,A -85,B 0,C 180,E1 -8253.295,E2 -8253.295} C_VEL
LIN {X 0,Y 453.507,Z 527.99,A -85,B 0,C 180,E1 -8256.24,E2 -8256.24} C_VEL
LIN {X 0,Y 453.488,Z 527.994,A -85,B 0,C 180,E1 -8259.118,E2 -8259.118} C_VEL
LIN {X 0,Y 453.509,Z 527.993,A -85,B 0,C 180,E1 -8261.945,E2 -8261.945} C_VEL
LIN {X 0,Y 453.546,Z 527.984,A -85,B 0,C 180,E1 -8264.727,E2 -8264.727} C_VEL
LIN {X 0,Y 453.565,Z 527.983,A -85,B 0,C 180,E1 -8268.38,E2 -8268.38} C_VEL
LIN {X 0,Y 453.658,Z 527.975,A -85,B 0,C 180,E1 -8271.986,E2 -8271.986} C_VEL
LIN {X 0,Y 453.675,Z 527.968,A -85,B 0,C 180,E1 -8274.667,E2 -8274.667} C_VEL
LIN {X 0,Y 453.75,Z 527.961,A -85,B 0,C 180,E1 -8277.337,E2 -8277.337} C_VEL
LIN {X 0,Y 453.83,Z 527.955,A -85,B 0,C 180,E1 -8280,E2 -8280} C_VEL
LIN {X 0,Y 453.751,Z 527.959,A -85,B 0,C 180,E1 -8282.664,E2 -8282.664} C_VEL
LIN {X 0,Y 453.684,Z 527.971,A -85,B 0,C 180,E1 -8286.226,E2 -8286.226} C_VEL
LIN {X 0,Y 453.598,Z 527.978,A -85,B 0,C 180,E1 -8288.914,E2 -8288.914} C_VEL
LIN {X 0,Y 453.571,Z 527.983,A -85,B 0,C 180,E1 -8292.529,E2 -8292.529} C_VEL
LIN {X 0,Y 453.552,Z 527.989,A -85,B 0,C 180,E1 -8296.196,E2 -8296.196} C_VEL
LIN {X 0,Y 453.525,Z 527.987,A -85,B 0,C 180,E1 -8299.039,E2 -8299.039} C_VEL
LIN {X 0,Y 453.484,Z 527.997,A -85,B 0,C 180,E1 -8301.836,E2 -8301.836} C_VEL
LIN {X 0,Y 453.509,Z 527.99,A -85,B 0,C 180,E1 -8304.735,E2 -8304.735} C_VEL
LIN {X 0,Y 453.54,Z 527.991,A -85,B 0,C 180,E1 -8307.959,E2 -8307.959} C_VEL
LIN {X 0,Y 453.473,Z 527.995,A -85,B 0,C 180,E1 -8311.525,E2 -8311.525} C_VEL
LIN {X 0,Y 453.495,Z 527.992,A -85,B 0,C 180,E1 -8314.777,E2 -8314.777} C_VEL
LIN {X 0,Y 453.468,Z 528.001,A -85,B 0,C 180,E1 -8318.312,E2 -8318.312} C_VEL
LIN {X 0,Y 453.501,Z 527.993,A -85,B 0,C 180,E1 -8320.609,E2 -8320.609} C_VEL
LIN {X 0,Y 453.467,Z 528.002,A -85,B 0,C 180,E1 -8324.221,E2 -8324.221} C_VEL
LIN {X 0,Y 453.47,Z 527.995,A -85,B 0,C 180,E1 -8327.005,E2 -8327.005} C_VEL
LIN {X 0,Y 453.524,Z 527.992,A -85,B 0,C 180,E1 -8330.553,E2 -8330.553} C_VEL
LIN {X 0,Y 453.461,Z 527.997,A -85,B 0,C 180,E1 -8333.917,E2 -8333.917} C_VEL
LIN {X 0,Y 453.49,Z 527.992,A -85,B 0,C 180,E1 -8337.151,E2 -8337.151} C_VEL
LIN {X 0,Y 453.482,Z 527.999,A -85,B 0,C 180,E1 -8340.268,E2 -8340.268} C_VEL
LIN {X 0,Y 453.522,Z 527.991,A -85,B 0,C 180,E1 -8343.294,E2 -8343.294} C_VEL
LIN {X 0,Y 453.585,Z 528.115,A -85,B 0,C 180,E1 -8343.786,E2 -8343.786} C_VEL
LIN {X 0,Y 455.651,Z 538.942,A -85,B 0,C 180,E1 -8345.99,E2 -8345.99} C_VEL
LIN {X 0,Y 456.037,Z 542.138,A -85,B 0,C 180,E1 -8346.618,E2 -8346.618} C_VEL
LIN {X 0,Y 455.175,Z 558.532,A -85,B 0,C 180,E1 -8349.67,E2 -8349.67} C_VEL
LIN {X 0,Y 454.458,Z 573.76,A -85,B 0,C 180,E1 -8352.466,E2 -8352.466} C_VEL
LIN {X 0,Y 457.595,Z 593.953,A -85,B 0,C 180,E1 -8352.922,E2 -8352.922} C_VEL
LIN {X 0,Y 456.787,Z 682.73,A -85,B 0,C 180,E1 -8354.379,E2 -8354.379} C_VEL
LIN {X 0,Y 456.352,Z 695.65,A -85,B 0,C 180,E1 -8354.764,E2 -8354.764} C_VEL
LIN {X 0,Y 455.859,Z 708.213,A -85,B 0,C 180,E1 -8355.319,E2 -8355.319} C_VEL
LIN {X 0,Y 455.301,Z 720.2,A -85,B 0,C 180,E1 -8356.042,E2 -8356.042} C_VEL
LIN {X 0,Y 454.737,Z 732.229,A -85,B 0,C 180,E1 -8356.983,E2 -8356.983} C_VEL
LIN {X 0,Y 454.274,Z 742.05,A -85,B 0,C 180,E1 -8357.943,E2 -8357.943} C_VEL
LIN {X 0,Y 453.703,Z 751.347,A -85,B 0,C 180,E1 -8359.06,E2 -8359.06} C_VEL
LIN {X 0,Y 453.249,Z 760.377,A -85,B 0,C 180,E1 -8360.404,E2 -8360.404} C_VEL
LIN {X 0,Y 452.939,Z 767.65,A -85,B 0,C 180,E1 -8361.747,E2 -8361.747} C_VEL
LIN {X 0,Y 452.725,Z 772.557,A -85,B 0,C 180,E1 -8362.865,E2 -8362.865} C_VEL
LIN {X 0,Y 452.585,Z 777.325,A -85,B 0,C 180,E1 -8364.206,E2 -8364.206} C_VEL
LIN {X 0,Y 452.492,Z 780.967,A -85,B 0,C 180,E1 -8365.545,E2 -8365.545} C_VEL
LIN {X 0,Y 452.483,Z 782.848,A -85,B 0,C 180,E1 -8366.437,E2 -8366.437} C_VEL
LIN {X 0,Y 452.509,Z 784.259,A -85,B 0,C 180,E1 -8367.328,E2 -8367.328} C_VEL
LIN {X 0,Y 452.429,Z 785.87,A -85,B 0,C 180,E1 -8369.109,E2 -8369.109} C_VEL
LIN {X 0,Y 452.434,Z 786.086,A -85,B 0,C 180,E1 -8369.999,E2 -8369.999} C_VEL
LIN {X 0,Y 452.428,Z 785.866,A -85,B 0,C 180,E1 -8370.889,E2 -8370.889} C_VEL
LIN {X 0,Y 452.508,Z 784.242,A -85,B 0,C 180,E1 -8372.669,E2 -8372.669} C_VEL
LIN {X 0,Y 452.483,Z 782.828,A -85,B 0,C 180,E1 -8373.561,E2 -8373.561} C_VEL
LIN {X 0,Y 452.552,Z 779.861,A -85,B 0,C 180,E1 -8374.898,E2 -8374.898} C_VEL
LIN {X 0,Y 452.628,Z 775.224,A -85,B 0,C 180,E1 -8376.415,E2 -8376.415} C_VEL
LIN {X 0,Y 452.869,Z 768.647,A -85,B 0,C 180,E1 -8378.027,E2 -8378.027} C_VEL
LIN {X 0,Y 453.199,Z 761.676,A -85,B 0,C 180,E1 -8379.37,E2 -8379.37} C_VEL
LIN {X 0,Y 453.601,Z 752.946,A -85,B 0,C 180,E1 -8380.714,E2 -8380.714} C_VEL
LIN {X 0,Y 454.157,Z 744.009,A -85,B 0,C 180,E1 -8381.831,E2 -8381.831} C_VEL
LIN {X 0,Y 454.659,Z 733.471,A -85,B 0,C 180,E1 -8382.907,E2 -8382.907} C_VEL
LIN {X 0,Y 455.29,Z 721.855,A -85,B 0,C 180,E1 -8383.842,E2 -8383.842} C_VEL
LIN {X 0,Y 455.827,Z 709.377,A -85,B 0,C 180,E1 -8384.622,E2 -8384.622} C_VEL
LIN {X 0,Y 456.341,Z 696.739,A -85,B 0,C 180,E1 -8385.205,E2 -8385.205} C_VEL
LIN {X 0,Y 456.791,Z 683.374,A -85,B 0,C 180,E1 -8385.618,E2 -8385.618} C_VEL
LIN {X 0,Y 457.122,Z 654.937,A -85,B 0,C 180,E1 -8386.108,E2 -8386.108} C_VEL
LIN {X 0,Y 457.554,Z 592.789,A -85,B 0,C 180,E1 -8387.123,E2 -8387.123} C_VEL
LIN {X 0,Y 454.454,Z 573.234,A -85,B 0,C 180,E1 -8387.596,E2 -8387.596} C_VEL
LIN {X 0,Y 455.187,Z 557.135,A -85,B 0,C 180,E1 -8390.563,E2 -8390.563} C_VEL
LIN {X 0,Y 456.035,Z 542.079,A -85,B 0,C 180,E1 -8393.379,E2 -8393.379} C_VEL
LIN {X 0,Y 455.131,Z 535.792,A -85,B 0,C 180,E1 -8394.639,E2 -8394.639} C_VEL
LIN {X 0,Y 453.533,Z 527.992,A -85,B 0,C 180,E1 -8396.31,E2 -8396.31} C_VEL
LIN {X 0,Y 453.509,Z 527.997,A -85,B 0,C 180,E1 -8398.71,E2 -8398.71} C_VEL
LIN {X 0,Y 453.462,Z 528.002,A -85,B 0,C 180,E1 -8401.798,E2 -8401.798} C_VEL
LIN {X 0,Y 453.477,Z 527.997,A -85,B 0,C 180,E1 -8404.988,E2 -8404.988} C_VEL
LIN {X 0,Y 453.48,Z 527.997,A -85,B 0,C 180,E1 -8408.308,E2 -8408.308} C_VEL
LIN {X 0,Y 453.511,Z 527.993,A -85,B 0,C 180,E1 -8410.605,E2 -8410.605} C_VEL
LIN {X 0,Y 453.467,Z 527.998,A -85,B 0,C 180,E1 -8414.219,E2 -8414.219} C_VEL
LIN {X 0,Y 453.456,Z 528.001,A -85,B 0,C 180,E1 -8417.004,E2 -8417.004} C_VEL
LIN {X 0,Y 453.524,Z 527.988,A -85,B 0,C 180,E1 -8420.553,E2 -8420.553} C_VEL
LIN {X 0,Y 453.45,Z 528,A -85,B 0,C 180,E1 -8423.916,E2 -8423.916} C_VEL
LIN {X 0,Y 453.475,Z 527.997,A -85,B 0,C 180,E1 -8427.15,E2 -8427.15} C_VEL
LIN {X 0,Y 453.505,Z 527.991,A -85,B 0,C 180,E1 -8430.27,E2 -8430.27} C_VEL
LIN {X 0,Y 453.505,Z 527.992,A -85,B 0,C 180,E1 -8433.293,E2 -8433.293} C_VEL
LIN {X 0,Y 453.494,Z 527.988,A -85,B 0,C 180,E1 -8436.238,E2 -8436.238} C_VEL
LIN {X 0,Y 453.473,Z 527.999,A -85,B 0,C 180,E1 -8439.117,E2 -8439.117} C_VEL
LIN {X 0,Y 453.502,Z 527.993,A -85,B 0,C 180,E1 -8441.944,E2 -8441.944} C_VEL
LIN {X 0,Y 453.53,Z 527.984,A -85,B 0,C 180,E1 -8444.726,E2 -8444.726} C_VEL
LIN {X 0,Y 453.591,Z 527.983,A -85,B 0,C 180,E1 -8447.471,E2 -8447.471} C_VEL
LIN {X 0,Y 453.582,Z 527.985,A -85,B 0,C 180,E1 -8451.086,E2 -8451.086} C_VEL
LIN {X 0,Y 453.667,Z 527.974,A -85,B 0,C 180,E1 -8453.774,E2 -8453.774} C_VEL
LIN {X 0,Y 453.756,Z 527.966,A -85,B 0,C 180,E1 -8457.336,E2 -8457.336} C_VEL
LIN {X 0,Y 453.813,Z 527.954,A -85,B 0,C 180,E1 -8460,E2 -8460} C_VEL
LIN {X 0,Y 453.756,Z 527.959,A -85,B 0,C 180,E1 -8462.663,E2 -8462.663} C_VEL
LIN {X 0,Y 453.671,Z 527.971,A -85,B 0,C 180,E1 -8466.225,E2 -8466.225} C_VEL
LIN {X 0,Y 453.582,Z 527.984,A -85,B 0,C 180,E1 -8468.913,E2 -8468.913} C_VEL
LIN {X 0,Y 453.589,Z 527.982,A -85,B 0,C 180,E1 -8472.551,E2 -8472.551} C_VEL
LIN {X 0,Y 453.532,Z 527.991,A -85,B 0,C 180,E1 -8476.196,E2 -8476.196} C_VEL
LIN {X 0,Y 453.508,Z 527.996,A -85,B 0,C 180,E1 -8479.041,E2 -8479.041} C_VEL
LIN {X 0,Y 453.464,Z 528.001,A -85,B 0,C 180,E1 -8481.836,E2 -8481.836} C_VEL
LIN {X 0,Y 453.502,Z 527.996,A -85,B 0,C 180,E1 -8484.735,E2 -8484.735} C_VEL
LIN {X 0,Y 453.571,Z 528.018,A -85,B 0,C 180,E1 -8487.512,E2 -8487.512} C_VEL
LIN {X 0,Y 455.144,Z 536.84,A -85,B 0,C 180,E1 -8489.611,E2 -8489.611} C_VEL
LIN {X 0,Y 454.772,Z 546.69,A -85,B 0,C 180,E1 -8491.795,E2 -8491.795} C_VEL
LIN {X 0,Y 454.655,Z 550.077,A -85,B 0,C 180,E1 -8492.501,E2 -8492.501} C_VEL
LIN {X 0,Y 457.821,Z 566.629,A -85,B 0,C 180,E1 -8492.91,E2 -8492.91} C_VEL
LIN {X 0,Y 456.876,Z 656.761,A -85,B 0,C 180,E1 -8494.392,E2 -8494.392} C_VEL
LIN {X 0,Y 456.555,Z 669.534,A -85,B 0,C 180,E1 -8494.77,E2 -8494.77} C_VEL
LIN {X 0,Y 456.137,Z 682.272,A -85,B 0,C 180,E1 -8495.329,E2 -8495.329} C_VEL
LIN {X 0,Y 455.66,Z 693.707,A -85,B 0,C 180,E1 -8496.007,E2 -8496.007} C_VEL
LIN {X 0,Y 455.072,Z 705.503,A -85,B 0,C 180,E1 -8496.917,E2 -8496.917} C_VEL
LIN {X 0,Y 454.528,Z 716.156,A -85,B 0,C 180,E1 -8497.95,E2 -8497.95} C_VEL
LIN {X 0,Y 454.023,Z 725.238,A -85,B 0,C 180,E1 -8499.04,E2 -8499.04} C_VEL
LIN {X 0,Y 453.541,Z 733.726,A -85,B 0,C 180,E1 -8500.295,E2 -8500.295} C_VEL
LIN {X 0,Y 453.159,Z 740.539,A -85,B 0,C 180,E1 -8501.529,E2 -8501.529} C_VEL
LIN {X 0,Y 452.884,Z 747.299,A -85,B 0,C 180,E1 -8503.063,E2 -8503.063} C_VEL
LIN {X 0,Y 452.661,Z 751.938,A -85,B 0,C 180,E1 -8504.425,E2 -8504.425} C_VEL
LIN {X 0,Y 452.5,Z 755.156,A -85,B 0,C 180,E1 -8505.662,E2 -8505.662} C_VEL
LIN {X 0,Y 452.423,Z 757.508,A -85,B 0,C 180,E1 -8506.894,E2 -8506.894} C_VEL
LIN {X 0,Y 452.319,Z 759.167,A -85,B 0,C 180,E1 -8508.228,E2 -8508.228} C_VEL
LIN {X 0,Y 452.297,Z 759.93,A -85,B 0,C 180,E1 -8509.586,E2 -8509.586} C_VEL
LIN {X 0,Y 452.295,Z 759.752,A -85,B 0,C 180,E1 -8510.979,E2 -8510.979} C_VEL
LIN {X 0,Y 452.365,Z 758.17,A -85,B 0,C 180,E1 -8512.708,E2 -8512.708} C_VEL
LIN {X 0,Y 452.555,Z 755.114,A -85,B 0,C 180,E1 -8514.404,E2 -8514.404} C_VEL
LIN {X 0,Y 452.68,Z 750.687,A -85,B 0,C 180,E1 -8516.021,E2 -8516.021} C_VEL
LIN {X 0,Y 452.911,Z 745.759,A -85,B 0,C 180,E1 -8517.371,E2 -8517.371} C_VEL
LIN {X 0,Y 453.232,Z 738.689,A -85,B 0,C 180,E1 -8518.888,E2 -8518.888} C_VEL
LIN {X 0,Y 453.704,Z 730.343,A -85,B 0,C 180,E1 -8520.287,E2 -8520.287} C_VEL
LIN {X 0,Y 454.162,Z 721.547,A -85,B 0,C 180,E1 -8521.481,E2 -8521.481} C_VEL
LIN {X 0,Y 454.312,Z 718.898,A -85,B 0,C 180,E1 -8521.793,E2 -8521.793} C_VEL
LIN {X 0,Y 453.896,Z 714.565,A -85,B 0,C 180,E1 -8522.291,E2 -8522.291} C_VEL
LIN {X 0,Y 451.498,Z 707.29,A -85,B 0,C 180,E1 -8523.085,E2 -8523.085} C_VEL
LIN {X 0,Y 449.09,Z 699.588,A -85,B 0,C 180,E1 -8523.816,E2 -8523.816} C_VEL
LIN {X 0,Y 448.663,Z 694.498,A -85,B 0,C 180,E1 -8524.211,E2 -8524.211} C_VEL
LIN {X 0,Y 449.176,Z 682.389,A -85,B 0,C 180,E1 -8524.95,E2 -8524.95} C_VEL
LIN {X 0,Y 449.65,Z 669.223,A -85,B 0,C 180,E1 -8525.533,E2 -8525.533} C_VEL
LIN {X 0,Y 449.987,Z 656.112,A -85,B 0,C 180,E1 -8525.921,E2 -8525.921} C_VEL
LIN {X 0,Y 450.929,Z 566.794,A -85,B 0,C 180,E1 -8527.403,E2 -8527.403} C_VEL
LIN {X 0,Y 447.569,Z 549.596,A -85,B 0,C 180,E1 -8527.832,E2 -8527.832} C_VEL
LIN {X 0,Y 448.067,Z 538.04,A -85,B 0,C 180,E1 -8530.394,E2 -8530.394} C_VEL
LIN {X 0,Y 446.51,Z 528.868,A -85,B 0,C 180,E1 -8532.601,E2 -8532.601} C_VEL
LIN {X 0,Y 446.467,Z 528.87,A -85,B 0,C 180,E1 -8535.414,E2 -8535.414} C_VEL
LIN {X 0,Y 446.513,Z 528.862,A -85,B 0,C 180,E1 -8538.194,E2 -8538.194} C_VEL
LIN {X 0,Y 446.596,Z 528.85,A -85,B 0,C 180,E1 -8541.859,E2 -8541.859} C_VEL
LIN {X 0,Y 446.639,Z 528.849,A -85,B 0,C 180,E1 -8544.584,E2 -8544.584} C_VEL
LIN {X 0,Y 446.707,Z 528.839,A -85,B 0,C 180,E1 -8547.296,E2 -8547.296} C_VEL
LIN {X 0,Y 446.791,Z 528.826,A -85,B 0,C 180,E1 -8550.001,E2 -8550.001} C_VEL
LIN {X 0,Y 446.706,Z 528.841,A -85,B 0,C 180,E1 -8552.707,E2 -8552.707} C_VEL
LIN {X 0,Y 446.637,Z 528.846,A -85,B 0,C 180,E1 -8556.325,E2 -8556.325} C_VEL
LIN {X 0,Y 446.536,Z 528.865,A -85,B 0,C 180,E1 -8559.057,E2 -8559.057} C_VEL
LIN {X 0,Y 446.521,Z 528.864,A -85,B 0,C 180,E1 -8562.731,E2 -8562.731} C_VEL
LIN {X 0,Y 446.495,Z 528.863,A -85,B 0,C 180,E1 -8566.229,E2 -8566.229} C_VEL
LIN {X 0,Y 446.468,Z 528.872,A -85,B 0,C 180,E1 -8569.304,E2 -8569.304} C_VEL
LIN {X 0,Y 446.418,Z 528.872,A -85,B 0,C 180,E1 -8572.201,E2 -8572.201} C_VEL
LIN {X 0,Y 446.458,Z 528.876,A -85,B 0,C 180,E1 -8575.153,E2 -8575.153} C_VEL
LIN {X 0,Y 446.485,Z 528.864,A -85,B 0,C 180,E1 -8578.18,E2 -8578.18} C_VEL
LIN {X 0,Y 446.42,Z 528.874,A -85,B 0,C 180,E1 -8581.776,E2 -8581.776} C_VEL
LIN {X 0,Y 446.43,Z 528.871,A -85,B 0,C 180,E1 -8584.524,E2 -8584.524} C_VEL
LIN {X 0,Y 446.417,Z 528.873,A -85,B 0,C 180,E1 -8588.08,E2 -8588.08} C_VEL
LIN {X 0,Y 446.43,Z 528.874,A -85,B 0,C 180,E1 -8590.919,E2 -8590.919} C_VEL
LIN {X 0,Y 446.426,Z 528.874,A -85,B 0,C 180,E1 -8593.844,E2 -8593.844} C_VEL
LIN {X 0,Y 446.402,Z 528.874,A -85,B 0,C 180,E1 -8596.404,E2 -8596.404} C_VEL
LIN {X 0,Y 446.43,Z 528.875,A -85,B 0,C 180,E1 -8599.083,E2 -8599.083} C_VEL
LIN {X 0,Y 446.413,Z 528.874,A -85,B 0,C 180,E1 -8602.122,E2 -8602.122} C_VEL
LIN {X 0,Y 446.433,Z 528.879,A -85,B 0,C 180,E1 -8605.478,E2 -8605.478} C_VEL
LIN {X 0,Y 446.42,Z 528.872,A -85,B 0,C 180,E1 -8608.701,E2 -8608.701} C_VEL
LIN {X 0,Y 446.489,Z 528.868,A -85,B 0,C 180,E1 -8611.822,E2 -8611.822} C_VEL
LIN {X 0,Y 446.454,Z 528.868,A -85,B 0,C 180,E1 -8614.848,E2 -8614.848} C_VEL
LIN {X 0,Y 446.453,Z 528.869,A -85,B 0,C 180,E1 -8618.246,E2 -8618.246} C_VEL
LIN {X 0,Y 446.458,Z 528.876,A -85,B 0,C 180,E1 -8621.65,E2 -8621.65} C_VEL
LIN {X 0,Y 446.514,Z 528.861,A -85,B 0,C 180,E1 -8624.48,E2 -8624.48} C_VEL
LIN {X 0,Y 446.523,Z 528.862,A -85,B 0,C 180,E1 -8628.194,E2 -8628.194} C_VEL
LIN {X 0,Y 446.607,Z 528.856,A -85,B 0,C 180,E1 -8631.858,E2 -8631.858} C_VEL
LIN {X 0,Y 446.649,Z 528.844,A -85,B 0,C 180,E1 -8634.583,E2 -8634.583} C_VEL
LIN {X 0,Y 446.671,Z 528.844,A -85,B 0,C 180,E1 -8638.197,E2 -8638.197} C_VEL
LIN {X 0,Y 446.8,Z 528.831,A -85,B 0,C 180,E1 -8640,E2 -8640} C_VEL
LIN {X 0,Y 446.697,Z 528.838,A -85,B 0,C 180,E1 -8642.706,E2 -8642.706} C_VEL
LIN {X 0,Y 446.654,Z 528.846,A -85,B 0,C 180,E1 -8646.324,E2 -8646.324} C_VEL
LIN {X 0,Y 446.544,Z 528.857,A -85,B 0,C 180,E1 -8649.056,E2 -8649.056} C_VEL
LIN {X 0,Y 446.529,Z 528.859,A -85,B 0,C 180,E1 -8652.73,E2 -8652.73} C_VEL
LIN {X 0,Y 446.503,Z 528.867,A -85,B 0,C 180,E1 -8656.228,E2 -8656.228} C_VEL
LIN {X 0,Y 446.476,Z 528.866,A -85,B 0,C 180,E1 -8659.303,E2 -8659.303} C_VEL
LIN {X 0,Y 446.426,Z 528.878,A -85,B 0,C 180,E1 -8662.2,E2 -8662.2} C_VEL
LIN {X 0,Y 446.452,Z 528.868,A -85,B 0,C 180,E1 -8665.153,E2 -8665.153} C_VEL
LIN {X 0,Y 446.493,Z 528.871,A -85,B 0,C 180,E1 -8668.179,E2 -8668.179} C_VEL
LIN {X 0,Y 446.426,Z 528.875,A -85,B 0,C 180,E1 -8671.775,E2 -8671.775} C_VEL
LIN {X 0,Y 446.437,Z 528.874,A -85,B 0,C 180,E1 -8674.523,E2 -8674.523} C_VEL
LIN {X 0,Y 446.421,Z 528.878,A -85,B 0,C 180,E1 -8678.079,E2 -8678.079} C_VEL
LIN {X 0,Y 446.429,Z 528.872,A -85,B 0,C 180,E1 -8680.916,E2 -8680.916} C_VEL
LIN {X 0,Y 446.405,Z 528.877,A -85,B 0,C 180,E1 -8683.846,E2 -8683.846} C_VEL
LIN {X 0,Y 446.406,Z 528.881,A -85,B 0,C 180,E1 -8686.403,E2 -8686.403} C_VEL
LIN {X 0,Y 446.434,Z 528.871,A -85,B 0,C 180,E1 -8689.082,E2 -8689.082} C_VEL
LIN {X 0,Y 446.437,Z 528.873,A -85,B 0,C 180,E1 -8691.918,E2 -8691.918} C_VEL
LIN {X 0,Y 446.436,Z 528.87,A -85,B 0,C 180,E1 -8695.476,E2 -8695.476} C_VEL
LIN {X 0,Y 446.423,Z 528.878,A -85,B 0,C 180,E1 -8698.699,E2 -8698.699} C_VEL
LIN {X 0,Y 446.492,Z 528.867,A -85,B 0,C 180,E1 -8701.821,E2 -8701.821} C_VEL
LIN {X 0,Y 446.533,Z 528.968,A -85,B 0,C 180,E1 -8703.556,E2 -8703.556} C_VEL
LIN {X 0,Y 448.771,Z 540.645,A -85,B 0,C 180,E1 -8705.971,E2 -8705.971} C_VEL
LIN {X 0,Y 449.04,Z 544.446,A -85,B 0,C 180,E1 -8706.721,E2 -8706.721} C_VEL
LIN {X 0,Y 448.084,Z 560.827,A -85,B 0,C 180,E1 -8709.813,E2 -8709.813} C_VEL
LIN {X 0,Y 447.485,Z 573.585,A -85,B 0,C 180,E1 -8712.194,E2 -8712.194} C_VEL
LIN {X 0,Y 450.741,Z 594.297,A -85,B 0,C 180,E1 -8712.672,E2 -8712.672} C_VEL
LIN {X 0,Y 449.912,Z 682.023,A -85,B 0,C 180,E1 -8714.134,E2 -8714.134} C_VEL
LIN {X 0,Y 449.497,Z 695.107,A -85,B 0,C 180,E1 -8714.526,E2 -8714.526} C_VEL
LIN {X 0,Y 449,Z 707.765,A -85,B 0,C 180,E1 -8715.09,E2 -8715.09} C_VEL
LIN {X 0,Y 448.411,Z 719.833,A -85,B 0,C 180,E1 -8715.823,E2 -8715.823} C_VEL
LIN {X 0,Y 447.822,Z 731.325,A -85,B 0,C 180,E1 -8716.727,E2 -8716.727} C_VEL
LIN {X 0,Y 447.295,Z 741.753,A -85,B 0,C 180,E1 -8717.752,E2 -8717.752} C_VEL
LIN {X 0,Y 446.702,Z 751.079,A -85,B 0,C 180,E1 -8718.887,E2 -8718.887} C_VEL
LIN {X 0,Y 446.221,Z 760.127,A -85,B 0,C 180,E1 -8720.251,E2 -8720.251} C_VEL
LIN {X 0,Y 445.866,Z 767.414,A -85,B 0,C 180,E1 -8721.615,E2 -8721.615} C_VEL
LIN {X 0,Y 445.646,Z 772.332,A -85,B 0,C 180,E1 -8722.751,E2 -8722.751} C_VEL
LIN {X 0,Y 445.496,Z 776.511,A -85,B 0,C 180,E1 -8723.925,E2 -8723.925} C_VEL
LIN {X 0,Y 445.418,Z 780.755,A -85,B 0,C 180,E1 -8725.474,E2 -8725.474} C_VEL
LIN {X 0,Y 445.382,Z 782.637,A -85,B 0,C 180,E1 -8726.38,E2 -8726.38} C_VEL
LIN {X 0,Y 445.434,Z 784.052,A -85,B 0,C 180,E1 -8727.286,E2 -8727.286} C_VEL
LIN {X 0,Y 445.339,Z 785.664,A -85,B 0,C 180,E1 -8729.094,E2 -8729.094} C_VEL
LIN {X 0,Y 445.342,Z 785.882,A -85,B 0,C 180,E1 -8729.999,E2 -8729.999} C_VEL
LIN {X 0,Y 445.339,Z 785.662,A -85,B 0,C 180,E1 -8730.903,E2 -8730.903} C_VEL
LIN {X 0,Y 445.433,Z 784.037,A -85,B 0,C 180,E1 -8732.712,E2 -8732.712} C_VEL
LIN {X 0,Y 445.381,Z 782.622,A -85,B 0,C 180,E1 -8733.618,E2 -8733.618} C_VEL
LIN {X 0,Y 445.481,Z 779.655,A -85,B 0,C 180,E1 -8734.976,E2 -8734.976} C_VEL
LIN {X 0,Y 445.576,Z 774.192,A -85,B 0,C 180,E1 -8736.747,E2 -8736.747} C_VEL
LIN {X 0,Y 445.802,Z 768.445,A -85,B 0,C 180,E1 -8738.155,E2 -8738.155} C_VEL
LIN {X 0,Y 446.148,Z 761.477,A -85,B 0,C 180,E1 -8739.519,E2 -8739.519} C_VEL
LIN {X 0,Y 446.589,Z 752.75,A -85,B 0,C 180,E1 -8740.884,E2 -8740.884} C_VEL
LIN {X 0,Y 447.203,Z 743.815,A -85,B 0,C 180,E1 -8742.017,E2 -8742.017} C_VEL
LIN {X 0,Y 447.752,Z 732.921,A -85,B 0,C 180,E1 -8743.143,E2 -8743.143} C_VEL
LIN {X 0,Y 448.371,Z 721.664,A -85,B 0,C 180,E1 -8744.06,E2 -8744.06} C_VEL
LIN {X 0,Y 448.958,Z 709.192,A -85,B 0,C 180,E1 -8744.851,E2 -8744.851} C_VEL
LIN {X 0,Y 449.488,Z 696.573,A -85,B 0,C 180,E1 -8745.442,E2 -8745.442} C_VEL
LIN {X 0,Y 449.967,Z 683.245,A -85,B 0,C 180,E1 -8745.861,E2 -8745.861} C_VEL
LIN {X 0,Y 450.264,Z 656.346,A -85,B 0,C 180,E1 -8746.337,E2 -8746.337} C_VEL
LIN {X 0,Y 450.827,Z 593.889,A -85,B 0,C 180,E1 -8747.37,E2 -8747.37} C_VEL
LIN {X 0,Y 447.522,Z 572.998,A -85,B 0,C 180,E1 -8747.89,E2 -8747.89} C_VEL
LIN {X 0,Y 448.321,Z 557,A -85,B 0,C 180,E1 -8750.892,E2 -8750.892} C_VEL
LIN {X 0,Y 449.098,Z 543.214,A -85,B 0,C 180,E1 -8753.517,E2 -8753.517} C_VEL
LIN {X 0,Y 447.911,Z 535.703,A -85,B 0,C 180,E1 -8755.063,E2 -8755.063} C_VEL
LIN {X 0,Y 446.483,Z 528.87,A -85,B 0,C 180,E1 -8756.549,E2 -8756.549} C_VEL
LIN {X 0,Y 446.447,Z 528.878,A -85,B 0,C 180,E1 -8759.208,E2 -8759.208} C_VEL
LIN {X 0,Y 446.419,Z 528.876,A -85,B 0,C 180,E1 -8762.36,E2 -8762.36} C_VEL
LIN {X 0,Y 446.417,Z 528.88,A -85,B 0,C 180,E1 -8765.624,E2 -8765.624} C_VEL
LIN {X 0,Y 446.47,Z 528.873,A -85,B 0,C 180,E1 -8769.022,E2 -8769.022} C_VEL
LIN {X 0,Y 446.432,Z 528.875,A -85,B 0,C 180,E1 -8772.276,E2 -8772.276} C_VEL
LIN {X 0,Y 446.448,Z 528.875,A -85,B 0,C 180,E1 -8775.102,E2 -8775.102} C_VEL
LIN {X 0,Y 446.428,Z 528.874,A -85,B 0,C 180,E1 -8778.608,E2 -8778.608} C_VEL
LIN {X 0,Y 446.466,Z 528.87,A -85,B 0,C 180,E1 -8780.975,E2 -8780.975} C_VEL
LIN {X 0,Y 446.414,Z 528.875,A -85,B 0,C 180,E1 -8784.373,E2 -8784.373} C_VEL
LIN {X 0,Y 446.415,Z 528.879,A -85,B 0,C 180,E1 -8787.637,E2 -8787.637} C_VEL
LIN {X 0,Y 446.461,Z 528.869,A -85,B 0,C 180,E1 -8790.791,E2 -8790.791} C_VEL
LIN {X 0,Y 446.468,Z 528.871,A -85,B 0,C 180,E1 -8793.847,E2 -8793.847} C_VEL
LIN {X 0,Y 446.419,Z 528.871,A -85,B 0,C 180,E1 -8796.822,E2 -8796.822} C_VEL
LIN {X 0,Y 446.435,Z 528.87,A -85,B 0,C 180,E1 -8799.736,E2 -8799.736} C_VEL
LIN {X 0,Y 446.453,Z 528.87,A -85,B 0,C 180,E1 -8802.596,E2 -8802.596} C_VEL
LIN {X 0,Y 446.461,Z 528.872,A -85,B 0,C 180,E1 -8805.412,E2 -8805.412} C_VEL
LIN {X 0,Y 446.529,Z 528.857,A -85,B 0,C 180,E1 -8808.193,E2 -8808.193} C_VEL
LIN {X 0,Y 446.589,Z 528.853,A -85,B 0,C 180,E1 -8811.857,E2 -8811.857} C_VEL
LIN {X 0,Y 446.636,Z 528.846,A -85,B 0,C 180,E1 -8814.582,E2 -8814.582} C_VEL
LIN {X 0,Y 446.7,Z 528.845,A -85,B 0,C 180,E1 -8817.294,E2 -8817.294} C_VEL
LIN {X 0,Y 446.783,Z 528.83,A -85,B 0,C 180,E1 -8820,E2 -8820} C_VEL
LIN {X 0,Y 446.7,Z 528.838,A -85,B 0,C 180,E1 -8822.705,E2 -8822.705} C_VEL
LIN {X 0,Y 446.64,Z 528.847,A -85,B 0,C 180,E1 -8826.323,E2 -8826.323} C_VEL
LIN {X 0,Y 446.528,Z 528.864,A -85,B 0,C 180,E1 -8829.055,E2 -8829.055} C_VEL
LIN {X 0,Y 446.522,Z 528.863,A -85,B 0,C 180,E1 -8832.729,E2 -8832.729} C_VEL
LIN {X 0,Y 446.477,Z 528.87,A -85,B 0,C 180,E1 -8836.459,E2 -8836.459} C_VEL
LIN {X 0,Y 446.457,Z 528.876,A -85,B 0,C 180,E1 -8839.303,E2 -8839.303} C_VEL
LIN {X 0,Y 446.405,Z 528.878,A -85,B 0,C 180,E1 -8842.2,E2 -8842.2} C_VEL
LIN {X 0,Y 446.446,Z 528.875,A -85,B 0,C 180,E1 -8845.152,E2 -8845.152} C_VEL
LIN {X 0,Y 446.516,Z 528.936,A -85,B 0,C 180,E1 -8847.284,E2 -8847.284} C_VEL
LIN {X 0,Y 448.223,Z 538.497,A -85,B 0,C 180,E1 -8849.597,E2 -8849.597} C_VEL
LIN {X 0,Y 447.687,Z 550.091,A -85,B 0,C 180,E1 -8852.202,E2 -8852.202} C_VEL
LIN {X 0,Y 451.078,Z 567.137,A -85,B 0,C 180,E1 -8852.644,E2 -8852.644} C_VEL
LIN {X 0,Y 450.053,Z 656.96,A -85,B 0,C 180,E1 -8854.145,E2 -8854.145} C_VEL
LIN {X 0,Y 449.73,Z 669.971,A -85,B 0,C 180,E1 -8854.539,E2 -8854.539} C_VEL
LIN {X 0,Y 449.3,Z 682.302,A -85,B 0,C 180,E1 -8855.088,E2 -8855.088} C_VEL
LIN {X 0,Y 448.798,Z 693.827,A -85,B 0,C 180,E1 -8855.78,E2 -8855.78} C_VEL
LIN {X 0,Y 448.184,Z 705.789,A -85,B 0,C 180,E1 -8856.716,E2 -8856.716} C_VEL
LIN {X 0,Y 447.562,Z 716.427,A -85,B 0,C 180,E1 -8857.763,E2 -8857.763} C_VEL
LIN {X 0,Y 447,Z 726.2,A -85,B 0,C 180,E1 -8858.969,E2 -8858.969} C_VEL
LIN {X 0,Y 446.472,Z 735.289,A -85,B 0,C 180,E1 -8860.365,E2 -8860.365} C_VEL
LIN {X 0,Y 446.02,Z 742.795,A -85,B 0,C 180,E1 -8861.818,E2 -8861.818} C_VEL
LIN {X 0,Y 445.809,Z 748.021,A -85,B 0,C 180,E1 -8863.086,E2 -8863.086} C_VEL
LIN {X 0,Y 445.512,Z 753.37,A -85,B 0,C 180,E1 -8864.777,E2 -8864.777} C_VEL
LIN {X 0,Y 445.362,Z 757.242,A -85,B 0,C 180,E1 -8866.543,E2 -8866.543} C_VEL
LIN {X 0,Y 445.261,Z 759.102,A -85,B 0,C 180,E1 -8867.888,E2 -8867.888} C_VEL
LIN {X 0,Y 445.199,Z 760.151,A -85,B 0,C 180,E1 -8869.669,E2 -8869.669} C_VEL
LIN {X 0,Y 445.221,Z 760.032,A -85,B 0,C 180,E1 -8870.847,E2 -8870.847} C_VEL
LIN {X 0,Y 445.253,Z 759.129,A -85,B 0,C 180,E1 -8872.111,E2 -8872.111} C_VEL
LIN {X 0,Y 445.349,Z 757.073,A -85,B 0,C 180,E1 -8873.592,E2 -8873.592} C_VEL
LIN {X 0,Y 445.495,Z 753.758,A -85,B 0,C 180,E1 -8875.118,E2 -8875.118} C_VEL
LIN {X 0,Y 445.711,Z 748.948,A -85,B 0,C 180,E1 -8876.689,E2 -8876.689} C_VEL
LIN {X 0,Y 445.949,Z 743.802,A -85,B 0,C 180,E1 -8877.989,E2 -8877.989} C_VEL
LIN {X 0,Y 446.352,Z 736.352,A -85,B 0,C 180,E1 -8879.485,E2 -8879.485} C_VEL
LIN {X 0,Y 446.821,Z 727.979,A -85,B 0,C 180,E1 -8880.819,E2 -8880.819} C_VEL
LIN {X 0,Y 447.35,Z 718.724,A -85,B 0,C 180,E1 -8882.01,E2 -8882.01} C_VEL
LIN {X 0,Y 447.875,Z 708.712,A -85,B 0,C 180,E1 -8883.059,E2 -8883.059} C_VEL
LIN {X 0,Y 448.504,Z 697.765,A -85,B 0,C 180,E1 -8883.977,E2 -8883.977} C_VEL
LIN {X 0,Y 448.663,Z 694.498,A -85,B 0,C 180,E1 -8884.211,E2 -8884.211} C_VEL
LIN {X 0,Y 448.214,Z 689.348,A -85,B 0,C 180,E1 -8884.582,E2 -8884.582} C_VEL
LIN {X 0,Y 445.725,Z 680.858,A -85,B 0,C 180,E1 -8885.167,E2 -8885.167} C_VEL
LIN {X 0,Y 443.272,Z 672.054,A -85,B 0,C 180,E1 -8885.657,E2 -8885.657} C_VEL
LIN {X 0,Y 442.863,Z 666.425,A -85,B 0,C 180,E1 -8885.875,E2 -8885.875} C_VEL
LIN {X 0,Y 443.185,Z 652.917,A -85,B 0,C 180,E1 -8886.227,E2 -8886.227} C_VEL
LIN {X 0,Y 444.113,Z 567.644,A -85,B 0,C 180,E1 -8887.656,E2 -8887.656} C_VEL
LIN {X 0,Y 440.644,Z 549.774,A -85,B 0,C 180,E1 -8888.112,E2 -8888.112} C_VEL
LIN {X 0,Y 441.105,Z 539.359,A -85,B 0,C 180,E1 -8890.454,E2 -8890.454} C_VEL
LIN {X 0,Y 439.462,Z 529.747,A -85,B 0,C 180,E1 -8892.793,E2 -8892.793} C_VEL
LIN {X 0,Y 439.429,Z 529.747,A -85,B 0,C 180,E1 -8896.121,E2 -8896.121} C_VEL
LIN {X 0,Y 439.433,Z 529.749,A -85,B 0,C 180,E1 -8898.937,E2 -8898.937} C_VEL
LIN {X 0,Y 439.595,Z 529.725,A -85,B 0,C 180,E1 -8902.398,E2 -8902.398} C_VEL
LIN {X 0,Y 439.614,Z 529.723,A -85,B 0,C 180,E1 -8904.497,E2 -8904.497} C_VEL
LIN {X 0,Y 439.633,Z 529.718,A -85,B 0,C 180,E1 -8908.169,E2 -8908.169} C_VEL
LIN {X 0,Y 439.761,Z 529.702,A -85,B 0,C 180,E1 -8910.001,E2 -8910.001} C_VEL
LIN {X 0,Y 439.653,Z 529.721,A -85,B 0,C 180,E1 -8912.75,E2 -8912.75} C_VEL
LIN {X 0,Y 439.609,Z 529.722,A -85,B 0,C 180,E1 -8916.427,E2 -8916.427} C_VEL
LIN {X 0,Y 439.498,Z 529.74,A -85,B 0,C 180,E1 -8919.203,E2 -8919.203} C_VEL
LIN {X 0,Y 439.465,Z 529.745,A -85,B 0,C 180,E1 -8922.939,E2 -8922.939} C_VEL
LIN {X 0,Y 439.446,Z 529.741,A -85,B 0,C 180,E1 -8926.35,E2 -8926.35} C_VEL
LIN {X 0,Y 439.402,Z 529.748,A -85,B 0,C 180,E1 -8929.628,E2 -8929.628} C_VEL
LIN {X 0,Y 439.365,Z 529.753,A -85,B 0,C 180,E1 -8932.577,E2 -8932.577} C_VEL
LIN {X 0,Y 439.405,Z 529.749,A -85,B 0,C 180,E1 -8935.586,E2 -8935.586} C_VEL
LIN {X 0,Y 439.418,Z 529.746,A -85,B 0,C 180,E1 -8938.675,E2 -8938.675} C_VEL
LIN {X 0,Y 439.371,Z 529.751,A -85,B 0,C 180,E1 -8942.032,E2 -8942.032} C_VEL
LIN {X 0,Y 439.396,Z 529.755,A -85,B 0,C 180,E1 -8945.341,E2 -8945.341} C_VEL
LIN {X 0,Y 439.385,Z 529.749,A -85,B 0,C 180,E1 -8948.596,E2 -8948.596} C_VEL
LIN {X 0,Y 439.392,Z 529.755,A -85,B 0,C 180,E1 -8951.258,E2 -8951.258} C_VEL
LIN {X 0,Y 439.408,Z 529.747,A -85,B 0,C 180,E1 -8954.73,E2 -8954.73} C_VEL
LIN {X 0,Y 439.399,Z 529.75,A -85,B 0,C 180,E1 -8957.797,E2 -8957.797} C_VEL
LIN {X 0,Y 439.429,Z 529.743,A -85,B 0,C 180,E1 -8960.228,E2 -8960.228} C_VEL
LIN {X 0,Y 439.377,Z 529.754,A -85,B 0,C 180,E1 -8963.714,E2 -8963.714} C_VEL
LIN {X 0,Y 439.376,Z 529.752,A -85,B 0,C 180,E1 -8967.055,E2 -8967.055} C_VEL
LIN {X 0,Y 439.386,Z 529.749,A -85,B 0,C 180,E1 -8970.275,E2 -8970.275} C_VEL
LIN {X 0,Y 439.433,Z 529.748,A -85,B 0,C 180,E1 -8973.397,E2 -8973.397} C_VEL
LIN {X 0,Y 439.391,Z 529.748,A -85,B 0,C 180,E1 -8976.43,E2 -8976.43} C_VEL
LIN {X 0,Y 439.394,Z 529.753,A -85,B 0,C 180,E1 -8979.398,E2 -8979.398} C_VEL
LIN {X 0,Y 439.412,Z 529.746,A -85,B 0,C 180,E1 -8982.309,E2 -8982.309} C_VEL
LIN {X 0,Y 439.454,Z 529.742,A -85,B 0,C 180,E1 -8985.175,E2 -8985.175} C_VEL
LIN {X 0,Y 439.489,Z 529.74,A -85,B 0,C 180,E1 -8988.002,E2 -8988.002} C_VEL
LIN {X 0,Y 439.554,Z 529.736,A -85,B 0,C 180,E1 -8991.727,E2 -8991.727} C_VEL
LIN {X 0,Y 439.625,Z 529.719,A -85,B 0,C 180,E1 -8994.496,E2 -8994.496} C_VEL
LIN {X 0,Y 439.641,Z 529.72,A -85,B 0,C 180,E1 -8998.168,E2 -8998.168} C_VEL
LIN {X 0,Y 439.769,Z 529.706,A -85,B 0,C 180,E1 -9000,E2 -9000} C_VEL
LIN {X 0,Y 439.647,Z 529.716,A -85,B 0,C 180,E1 -9002.749,E2 -9002.749} C_VEL
LIN {X 0,Y 439.625,Z 529.72,A -85,B 0,C 180,E1 -9006.426,E2 -9006.426} C_VEL
LIN {X 0,Y 439.506,Z 529.734,A -85,B 0,C 180,E1 -9009.202,E2 -9009.202} C_VEL
LIN {X 0,Y 439.473,Z 529.737,A -85,B 0,C 180,E1 -9012.938,E2 -9012.938} C_VEL
LIN {X 0,Y 439.454,Z 529.743,A -85,B 0,C 180,E1 -9016.348,E2 -9016.348} C_VEL
LIN {X 0,Y 439.41,Z 529.748,A -85,B 0,C 180,E1 -9019.626,E2 -9019.626} C_VEL
LIN {X 0,Y 439.372,Z 529.752,A -85,B 0,C 180,E1 -9022.576,E2 -9022.576} C_VEL
LIN {X 0,Y 439.405,Z 529.748,A -85,B 0,C 180,E1 -9025.585,E2 -9025.585} C_VEL
LIN {X 0,Y 439.425,Z 529.745,A -85,B 0,C 180,E1 -9028.673,E2 -9028.673} C_VEL
LIN {X 0,Y 439.377,Z 529.756,A -85,B 0,C 180,E1 -9032.03,E2 -9032.03} C_VEL
LIN {X 0,Y 439.403,Z 529.746,A -85,B 0,C 180,E1 -9035.34,E2 -9035.34} C_VEL
LIN {X 0,Y 439.378,Z 529.753,A -85,B 0,C 180,E1 -9038.596,E2 -9038.596} C_VEL
LIN {X 0,Y 439.388,Z 529.748,A -85,B 0,C 180,E1 -9041.255,E2 -9041.255} C_VEL
LIN {X 0,Y 439.406,Z 529.748,A -85,B 0,C 180,E1 -9044.729,E2 -9044.729} C_VEL
LIN {X 0,Y 439.403,Z 529.748,A -85,B 0,C 180,E1 -9047.795,E2 -9047.795} C_VEL
LIN {X 0,Y 439.444,Z 529.748,A -85,B 0,C 180,E1 -9050.228,E2 -9050.228} C_VEL
LIN {X 0,Y 439.381,Z 529.75,A -85,B 0,C 180,E1 -9053.712,E2 -9053.712} C_VEL
LIN {X 0,Y 439.379,Z 529.75,A -85,B 0,C 180,E1 -9057.053,E2 -9057.053} C_VEL
LIN {X 0,Y 439.389,Z 529.754,A -85,B 0,C 180,E1 -9060.273,E2 -9060.273} C_VEL
LIN {X 0,Y 439.465,Z 529.901,A -85,B 0,C 180,E1 -9063.333,E2 -9063.333} C_VEL
LIN {X 0,Y 441.554,Z 540.403,A -85,B 0,C 180,E1 -9065.553,E2 -9065.553} C_VEL
LIN {X 0,Y 442.103,Z 545.475,A -85,B 0,C 180,E1 -9066.582,E2 -9066.582} C_VEL
LIN {X 0,Y 441.206,Z 560.6,A -85,B 0,C 180,E1 -9069.485,E2 -9069.485} C_VEL
LIN {X 0,Y 440.539,Z 573.394,A -85,B 0,C 180,E1 -9071.912,E2 -9071.912} C_VEL
LIN {X 0,Y 443.948,Z 595.668,A -85,B 0,C 180,E1 -9072.436,E2 -9072.436} C_VEL
LIN {X 0,Y 443.062,Z 681.314,A -85,B 0,C 180,E1 -9073.882,E2 -9073.882} C_VEL
LIN {X 0,Y 442.634,Z 694.563,A -85,B 0,C 180,E1 -9074.28,E2 -9074.28} C_VEL
LIN {X 0,Y 442.134,Z 707.308,A -85,B 0,C 180,E1 -9074.853,E2 -9074.853} C_VEL
LIN {X 0,Y 441.518,Z 719.452,A -85,B 0,C 180,E1 -9075.597,E2 -9075.597} C_VEL
LIN {X 0,Y 440.877,Z 730.914,A -85,B 0,C 180,E1 -9076.508,E2 -9076.508} C_VEL
LIN {X 0,Y 440.313,Z 741.431,A -85,B 0,C 180,E1 -9077.555,E2 -9077.555} C_VEL
LIN {X 0,Y 439.718,Z 750.789,A -85,B 0,C 180,E1 -9078.708,E2 -9078.708} C_VEL
LIN {X 0,Y 439.199,Z 759.853,A -85,B 0,C 180,E1 -9080.093,E2 -9080.093} C_VEL
LIN {X 0,Y 438.812,Z 767.154,A -85,B 0,C 180,E1 -9081.479,E2 -9081.479} C_VEL
LIN {X 0,Y 438.594,Z 772.085,A -85,B 0,C 180,E1 -9082.634,E2 -9082.634} C_VEL
LIN {X 0,Y 438.395,Z 776.709,A -85,B 0,C 180,E1 -9083.966,E2 -9083.966} C_VEL
LIN {X 0,Y 438.347,Z 780.53,A -85,B 0,C 180,E1 -9085.401,E2 -9085.401} C_VEL
LIN {X 0,Y 438.284,Z 782.417,A -85,B 0,C 180,E1 -9086.321,E2 -9086.321} C_VEL
LIN {X 0,Y 438.342,Z 783.838,A -85,B 0,C 180,E1 -9087.242,E2 -9087.242} C_VEL
LIN {X 0,Y 438.252,Z 785.456,A -85,B 0,C 180,E1 -9089.08,E2 -9089.08} C_VEL
LIN {X 0,Y 438.253,Z 785.677,A -85,B 0,C 180,E1 -9089.999,E2 -9089.999} C_VEL
LIN {X 0,Y 438.252,Z 785.46,A -85,B 0,C 180,E1 -9090.918,E2 -9090.918} C_VEL
LIN {X 0,Y 438.341,Z 783.838,A -85,B 0,C 180,E1 -9092.756,E2 -9092.756} C_VEL
LIN {X 0,Y 438.283,Z 782.424,A -85,B 0,C 180,E1 -9093.676,E2 -9093.676} C_VEL
LIN {X 0,Y 438.391,Z 779.458,A -85,B 0,C 180,E1 -9095.057,E2 -9095.057} C_VEL
LIN {X 0,Y 438.449,Z 775.442,A -85,B 0,C 180,E1 -9096.441,E2 -9096.441} C_VEL
LIN {X 0,Y 438.697,Z 769.269,A -85,B 0,C 180,E1 -9098.057,E2 -9098.057} C_VEL
LIN {X 0,Y 439.056,Z 762.528,A -85,B 0,C 180,E1 -9099.442,E2 -9099.442} C_VEL
LIN {X 0,Y 439.501,Z 754.166,A -85,B 0,C 180,E1 -9100.828,E2 -9100.828} C_VEL
LIN {X 0,Y 440.099,Z 745.584,A -85,B 0,C 180,E1 -9101.98,E2 -9101.98} C_VEL
LIN {X 0,Y 440.636,Z 735.466,A -85,B 0,C 180,E1 -9103.088,E2 -9103.088} C_VEL
LIN {X 0,Y 441.322,Z 724.501,A -85,B 0,C 180,E1 -9104.054,E2 -9104.054} C_VEL
LIN {X 0,Y 441.882,Z 712.978,A -85,B 0,C 180,E1 -9104.859,E2 -9104.859} C_VEL
LIN {X 0,Y 442.536,Z 699.764,A -85,B 0,C 180,E1 -9105.544,E2 -9105.544} C_VEL
LIN {X 0,Y 443.023,Z 686.454,A -85,B 0,C 180,E1 -9106.028,E2 -9106.028} C_VEL
LIN {X 0,Y 443.355,Z 671.595,A -85,B 0,C 180,E1 -9106.341,E2 -9106.341} C_VEL
LIN {X 0,Y 444.025,Z 594.496,A -85,B 0,C 180,E1 -9107.642,E2 -9107.642} C_VEL
LIN {X 0,Y 440.587,Z 572.779,A -85,B 0,C 180,E1 -9108.197,E2 -9108.197} C_VEL
LIN {X 0,Y 441.476,Z 555.612,A -85,B 0,C 180,E1 -9111.476,E2 -9111.476} C_VEL
LIN {X 0,Y 442.159,Z 544.363,A -85,B 0,C 180,E1 -9113.66,E2 -9113.66} C_VEL
LIN {X 0,Y 440.672,Z 535.618,A -85,B 0,C 180,E1 -9115.504,E2 -9115.504} C_VEL
LIN {X 0,Y 439.443,Z 529.748,A -85,B 0,C 180,E1 -9116.793,E2 -9116.793} C_VEL
LIN {X 0,Y 439.381,Z 529.76,A -85,B 0,C 180,E1 -9119.724,E2 -9119.724} C_VEL
LIN {X 0,Y 439.369,Z 529.754,A -85,B 0,C 180,E1 -9122.944,E2 -9122.944} C_VEL
LIN {X 0,Y 439.373,Z 529.754,A -85,B 0,C 180,E1 -9126.285,E2 -9126.285} C_VEL
LIN {X 0,Y 439.423,Z 529.751,A -85,B 0,C 180,E1 -9129.852,E2 -9129.852} C_VEL
LIN {X 0,Y 439.38,Z 529.753,A -85,B 0,C 180,E1 -9132.626,E2 -9132.626} C_VEL
LIN {X 0,Y 439.396,Z 529.755,A -85,B 0,C 180,E1 -9135.269,E2 -9135.269} C_VEL
LIN {X 0,Y 439.391,Z 529.751,A -85,B 0,C 180,E1 -9138.74,E2 -9138.74} C_VEL
LIN {X 0,Y 439.384,Z 529.754,A -85,B 0,C 180,E1 -9141.603,E2 -9141.603} C_VEL
LIN {X 0,Y 439.393,Z 529.751,A -85,B 0,C 180,E1 -9144.843,E2 -9144.843} C_VEL
LIN {X 0,Y 439.366,Z 529.752,A -85,B 0,C 180,E1 -9148.139,E2 -9148.139} C_VEL
LIN {X 0,Y 439.416,Z 529.752,A -85,B 0,C 180,E1 -9151.326,E2 -9151.326} C_VEL
LIN {X 0,Y 439.396,Z 529.749,A -85,B 0,C 180,E1 -9154.414,E2 -9154.414} C_VEL
LIN {X 0,Y 439.355,Z 529.756,A -85,B 0,C 180,E1 -9157.424,E2 -9157.424} C_VEL
LIN {X 0,Y 439.431,Z 529.739,A -85,B 0,C 180,E1 -9160.662,E2 -9160.662} C_VEL
LIN {X 0,Y 439.452,Z 529.737,A -85,B 0,C 180,E1 -9164.224,E2 -9164.224} C_VEL
LIN {X 0,Y 439.497,Z 529.734,A -85,B 0,C 180,E1 -9168.001,E2 -9168.001} C_VEL
LIN {X 0,Y 439.537,Z 529.731,A -85,B 0,C 180,E1 -9171.726,E2 -9171.726} C_VEL
LIN {X 0,Y 439.611,Z 529.721,A -85,B 0,C 180,E1 -9174.495,E2 -9174.495} C_VEL
LIN {X 0,Y 439.625,Z 529.718,A -85,B 0,C 180,E1 -9178.167,E2 -9178.167} C_VEL
LIN {X 0,Y 439.753,Z 529.706,A -85,B 0,C 180,E1 -9180,E2 -9180} C_VEL
LIN {X 0,Y 439.647,Z 529.717,A -85,B 0,C 180,E1 -9182.748,E2 -9182.748} C_VEL
LIN {X 0,Y 439.61,Z 529.723,A -85,B 0,C 180,E1 -9186.425,E2 -9186.425} C_VEL
LIN {X 0,Y 439.49,Z 529.743,A -85,B 0,C 180,E1 -9189.201,E2 -9189.201} C_VEL
LIN {X 0,Y 439.492,Z 529.739,A -85,B 0,C 180,E1 -9192.727,E2 -9192.727} C_VEL
LIN {X 0,Y 439.435,Z 529.747,A -85,B 0,C 180,E1 -9196.349,E2 -9196.349} C_VEL
LIN {X 0,Y 439.39,Z 529.755,A -85,B 0,C 180,E1 -9199.626,E2 -9199.626} C_VEL
LIN {X 0,Y 439.352,Z 529.757,A -85,B 0,C 180,E1 -9202.576,E2 -9202.576} C_VEL
LIN {X 0,Y 439.393,Z 529.755,A -85,B 0,C 180,E1 -9205.585,E2 -9205.585} C_VEL
LIN {X 0,Y 439.467,Z 529.863,A -85,B 0,C 180,E1 -9207.05,E2 -9207.05} C_VEL
LIN {X 0,Y 441.229,Z 539.067,A -85,B 0,C 180,E1 -9209.326,E2 -9209.326} C_VEL
LIN {X 0,Y 440.953,Z 547.212,A -85,B 0,C 180,E1 -9211.197,E2 -9211.197} C_VEL
LIN {X 0,Y 440.835,Z 550.591,A -85,B 0,C 180,E1 -9211.909,E2 -9211.909} C_VEL
LIN {X 0,Y 444.328,Z 568.489,A -85,B 0,C 180,E1 -9212.378,E2 -9212.378} C_VEL
LIN {X 0,Y 443.234,Z 657.507,A -85,B 0,C 180,E1 -9213.898,E2 -9213.898} C_VEL
LIN {X 0,Y 442.919,Z 670.262,A -85,B 0,C 180,E1 -9214.293,E2 -9214.293} C_VEL
LIN {X 0,Y 442.464,Z 681.749,A -85,B 0,C 180,E1 -9214.808,E2 -9214.808} C_VEL
LIN {X 0,Y 441.994,Z 692.924,A -85,B 0,C 180,E1 -9215.476,E2 -9215.476} C_VEL
LIN {X 0,Y 441.4,Z 704.583,A -85,B 0,C 180,E1 -9216.376,E2 -9216.376} C_VEL
LIN {X 0,Y 440.8,Z 714.091,A -85,B 0,C 180,E1 -9217.29,E2 -9217.29} C_VEL
LIN {X 0,Y 440.149,Z 724.462,A -85,B 0,C 180,E1 -9218.522,E2 -9218.522} C_VEL
LIN {X 0,Y 439.636,Z 732.815,A -85,B 0,C 180,E1 -9219.749,E2 -9219.749} C_VEL
LIN {X 0,Y 439.104,Z 740.815,A -85,B 0,C 180,E1 -9221.217,E2 -9221.217} C_VEL
LIN {X 0,Y 438.794,Z 746.618,A -85,B 0,C 180,E1 -9222.546,E2 -9222.546} C_VEL
LIN {X 0,Y 438.585,Z 751.201,A -85,B 0,C 180,E1 -9223.858,E2 -9223.858} C_VEL
LIN {X 0,Y 438.369,Z 754.717,A -85,B 0,C 180,E1 -9225.139,E2 -9225.139} C_VEL
LIN {X 0,Y 438.291,Z 757.34,A -85,B 0,C 180,E1 -9226.411,E2 -9226.411} C_VEL
LIN {X 0,Y 438.197,Z 759.089,A -85,B 0,C 180,E1 -9227.656,E2 -9227.656} C_VEL
LIN {X 0,Y 438.127,Z 760.113,A -85,B 0,C 180,E1 -9228.931,E2 -9228.931} C_VEL
LIN {X 0,Y 438.107,Z 760.358,A -85,B 0,C 180,E1 -9230.353,E2 -9230.353} C_VEL
LIN {X 0,Y 438.151,Z 759.621,A -85,B 0,C 180,E1 -9231.809,E2 -9231.809} C_VEL
LIN {X 0,Y 438.259,Z 757.328,A -85,B 0,C 180,E1 -9233.608,E2 -9233.608} C_VEL
LIN {X 0,Y 438.447,Z 753.492,A -85,B 0,C 180,E1 -9235.362,E2 -9235.362} C_VEL
LIN {X 0,Y 438.676,Z 748.405,A -85,B 0,C 180,E1 -9236.997,E2 -9236.997} C_VEL
LIN {X 0,Y 438.997,Z 742.794,A -85,B 0,C 180,E1 -9238.381,E2 -9238.381} C_VEL
LIN {X 0,Y 439.37,Z 735.915,A -85,B 0,C 180,E1 -9239.741,E2 -9239.741} C_VEL
LIN {X 0,Y 439.885,Z 727.322,A -85,B 0,C 180,E1 -9241.1,E2 -9241.1} C_VEL
LIN {X 0,Y 440.472,Z 717.883,A -85,B 0,C 180,E1 -9242.31,E2 -9242.31} C_VEL
LIN {X 0,Y 441.098,Z 707.744,A -85,B 0,C 180,E1 -9243.363,E2 -9243.363} C_VEL
LIN {X 0,Y 441.691,Z 696.302,A -85,B 0,C 180,E1 -9244.306,E2 -9244.306} C_VEL
LIN {X 0,Y 442.197,Z 684.751,A -85,B 0,C 180,E1 -9245.054,E2 -9245.054} C_VEL
LIN {X 0,Y 442.679,Z 673.123,A -85,B 0,C 180,E1 -9245.622,E2 -9245.622} C_VEL
LIN {X 0,Y 442.863,Z 666.425,A -85,B 0,C 180,E1 -9245.875,E2 -9245.875} C_VEL
LIN {X 0,Y 442.513,Z 660.711,A -85,B 0,C 180,E1 -9246.067,E2 -9246.067} C_VEL
LIN {X 0,Y 437.165,Z 642.107,A -85,B 0,C 180,E1 -9246.644,E2 -9246.644} C_VEL
LIN {X 0,Y 436.527,Z 636.295,A -85,B 0,C 180,E1 -9246.765,E2 -9246.765} C_VEL
LIN {X 0,Y 437.226,Z 567.824,A -85,B 0,C 180,E1 -9247.932,E2 -9247.932} C_VEL
LIN {X 0,Y 433.719,Z 549.959,A -85,B 0,C 180,E1 -9248.401,E2 -9248.401} C_VEL
LIN {X 0,Y 434.113,Z 540.238,A -85,B 0,C 180,E1 -9250.619,E2 -9250.619} C_VEL
LIN {X 0,Y 432.437,Z 530.621,A -85,B 0,C 180,E1 -9252.992,E2 -9252.992} C_VEL
LIN {X 0,Y 432.377,Z 530.625,A -85,B 0,C 180,E1 -9255.89,E2 -9255.89} C_VEL
LIN {X 0,Y 432.389,Z 530.628,A -85,B 0,C 180,E1 -9258.754,E2 -9258.754} C_VEL
LIN {X 0,Y 432.555,Z 530.601,A -85,B 0,C 180,E1 -9262.348,E2 -9262.348} C_VEL
LIN {X 0,Y 432.59,Z 530.597,A -85,B 0,C 180,E1 -9264.407,E2 -9264.407} C_VEL
LIN {X 0,Y 432.603,Z 530.594,A -85,B 0,C 180,E1 -9268.139,E2 -9268.139} C_VEL
LIN {X 0,Y 432.731,Z 530.577,A -85,B 0,C 180,E1 -9270.001,E2 -9270.001} C_VEL
LIN {X 0,Y 432.602,Z 530.599,A -85,B 0,C 180,E1 -9272.795,E2 -9272.795} C_VEL
LIN {X 0,Y 432.562,Z 530.601,A -85,B 0,C 180,E1 -9276.532,E2 -9276.532} C_VEL
LIN {X 0,Y 432.441,Z 530.617,A -85,B 0,C 180,E1 -9279.354,E2 -9279.354} C_VEL
LIN {X 0,Y 432.43,Z 530.62,A -85,B 0,C 180,E1 -9282.805,E2 -9282.805} C_VEL
LIN {X 0,Y 432.411,Z 530.619,A -85,B 0,C 180,E1 -9286.48,E2 -9286.48} C_VEL
LIN {X 0,Y 432.338,Z 530.627,A -85,B 0,C 180,E1 -9289.962,E2 -9289.962} C_VEL
LIN {X 0,Y 432.319,Z 530.634,A -85,B 0,C 180,E1 -9292.965,E2 -9292.965} C_VEL
LIN {X 0,Y 432.365,Z 530.623,A -85,B 0,C 180,E1 -9296.034,E2 -9296.034} C_VEL
LIN {X 0,Y 432.344,Z 530.634,A -85,B 0,C 180,E1 -9299.189,E2 -9299.189} C_VEL
LIN {X 0,Y 432.324,Z 530.628,A -85,B 0,C 180,E1 -9302.444,E2 -9302.444} C_VEL
LIN {X 0,Y 432.346,Z 530.629,A -85,B 0,C 180,E1 -9305.633,E2 -9305.633} C_VEL
LIN {X 0,Y 432.352,Z 530.632,A -85,B 0,C 180,E1 -9309.344,E2 -9309.344} C_VEL
LIN {X 0,Y 432.338,Z 530.629,A -85,B 0,C 180,E1 -9311.798,E2 -9311.798} C_VEL
LIN {X 0,Y 432.343,Z 530.626,A -85,B 0,C 180,E1 -9314.347,E2 -9314.347} C_VEL
LIN {X 0,Y 432.323,Z 530.631,A -85,B 0,C 180,E1 -9317.017,E2 -9317.017} C_VEL
LIN {X 0,Y 432.336,Z 530.63,A -85,B 0,C 180,E1 -9319.822,E2 -9319.822} C_VEL
LIN {X 0,Y 432.31,Z 530.633,A -85,B 0,C 180,E1 -9323.023,E2 -9323.023} C_VEL
LIN {X 0,Y 432.363,Z 530.625,A -85,B 0,C 180,E1 -9325.997,E2 -9325.997} C_VEL
LIN {X 0,Y 432.352,Z 530.633,A -85,B 0,C 180,E1 -9329.491,E2 -9329.491} C_VEL
LIN {X 0,Y 432.396,Z 530.62,A -85,B 0,C 180,E1 -9332.929,E2 -9332.929} C_VEL
LIN {X 0,Y 432.375,Z 530.624,A -85,B 0,C 180,E1 -9336.024,E2 -9336.024} C_VEL
LIN {X 0,Y 432.355,Z 530.626,A -85,B 0,C 180,E1 -9339.047,E2 -9339.047} C_VEL
LIN {X 0,Y 432.367,Z 530.626,A -85,B 0,C 180,E1 -9342.011,E2 -9342.011} C_VEL
LIN {X 0,Y 432.401,Z 530.619,A -85,B 0,C 180,E1 -9344.927,E2 -9344.927} C_VEL
LIN {X 0,Y 432.465,Z 530.617,A -85,B 0,C 180,E1 -9347.804,E2 -9347.804} C_VEL
LIN {X 0,Y 432.498,Z 530.612,A -85,B 0,C 180,E1 -9351.591,E2 -9351.591} C_VEL
LIN {X 0,Y 432.601,Z 530.595,A -85,B 0,C 180,E1 -9354.407,E2 -9354.407} C_VEL
LIN {X 0,Y 432.61,Z 530.596,A -85,B 0,C 180,E1 -9358.139,E2 -9358.139} C_VEL
LIN {X 0,Y 432.739,Z 530.582,A -85,B 0,C 180,E1 -9360,E2 -9360} C_VEL
LIN {X 0,Y 432.599,Z 530.594,A -85,B 0,C 180,E1 -9362.794,E2 -9362.794} C_VEL
LIN {X 0,Y 432.58,Z 530.597,A -85,B 0,C 180,E1 -9366.531,E2 -9366.531} C_VEL
LIN {X 0,Y 432.449,Z 530.614,A -85,B 0,C 180,E1 -9369.353,E2 -9369.353} C_VEL
LIN {X 0,Y 432.439,Z 530.614,A -85,B 0,C 180,E1 -9372.804,E2 -9372.804} C_VEL
LIN {X 0,Y 432.42,Z 530.618,A -85,B 0,C 180,E1 -9376.479,E2 -9376.479} C_VEL
LIN {X 0,Y 432.347,Z 530.633,A -85,B 0,C 180,E1 -9379.961,E2 -9379.961} C_VEL
LIN {X 0,Y 432.326,Z 530.628,A -85,B 0,C 180,E1 -9382.964,E2 -9382.964} C_VEL
LIN {X 0,Y 432.369,Z 530.63,A -85,B 0,C 180,E1 -9386.033,E2 -9386.033} C_VEL
LIN {X 0,Y 432.351,Z 530.625,A -85,B 0,C 180,E1 -9389.187,E2 -9389.187} C_VEL
LIN {X 0,Y 432.33,Z 530.632,A -85,B 0,C 180,E1 -9392.443,E2 -9392.443} C_VEL
LIN {X 0,Y 432.352,Z 530.626,A -85,B 0,C 180,E1 -9395.632,E2 -9395.632} C_VEL
LIN {X 0,Y 432.341,Z 530.628,A -85,B 0,C 180,E1 -9398.713,E2 -9398.713} C_VEL
LIN {X 0,Y 432.331,Z 530.63,A -85,B 0,C 180,E1 -9401.798,E2 -9401.798} C_VEL
LIN {X 0,Y 432.341,Z 530.633,A -85,B 0,C 180,E1 -9404.347,E2 -9404.347} C_VEL
LIN {X 0,Y 432.327,Z 530.628,A -85,B 0,C 180,E1 -9407.015,E2 -9407.015} C_VEL
LIN {X 0,Y 432.348,Z 530.627,A -85,B 0,C 180,E1 -9409.819,E2 -9409.819} C_VEL
LIN {X 0,Y 432.318,Z 530.63,A -85,B 0,C 180,E1 -9413.022,E2 -9413.022} C_VEL
LIN {X 0,Y 432.366,Z 530.626,A -85,B 0,C 180,E1 -9415.996,E2 -9415.996} C_VEL
LIN {X 0,Y 432.355,Z 530.627,A -85,B 0,C 180,E1 -9419.489,E2 -9419.489} C_VEL
LIN {X 0,Y 432.434,Z 530.62,A -85,B 0,C 180,E1 -9423.06,E2 -9423.06} C_VEL
LIN {X 0,Y 434.753,Z 542.698,A -85,B 0,C 180,E1 -9425.654,E2 -9425.654} C_VEL
LIN {X 0,Y 435.168,Z 546.627,A -85,B 0,C 180,E1 -9426.464,E2 -9426.464} C_VEL
LIN {X 0,Y 434.063,Z 564.263,A -85,B 0,C 180,E1 -9429.9,E2 -9429.9} C_VEL
LIN {X 0,Y 433.591,Z 573.198,A -85,B 0,C 180,E1 -9431.622,E2 -9431.622} C_VEL
LIN {X 0,Y 437.146,Z 596.735,A -85,B 0,C 180,E1 -9432.186,E2 -9432.186} C_VEL
LIN {X 0,Y 436.216,Z 681.745,A -85,B 0,C 180,E1 -9433.652,E2 -9433.652} C_VEL
LIN {X 0,Y 435.733,Z 695.535,A -85,B 0,C 180,E1 -9434.085,E2 -9434.085} C_VEL
LIN {X 0,Y 435.218,Z 707.961,A -85,B 0,C 180,E1 -9434.666,E2 -9434.666} C_VEL
LIN {X 0,Y 434.621,Z 719.07,A -85,B 0,C 180,E1 -9435.364,E2 -9435.364} C_VEL
LIN {X 0,Y 433.951,Z 730.443,A -85,B 0,C 180,E1 -9436.278,E2 -9436.278} C_VEL
LIN {X 0,Y 433.333,Z 741.109,A -85,B 0,C 180,E1 -9437.351,E2 -9437.351} C_VEL
LIN {X 0,Y 432.742,Z 750.498,A -85,B 0,C 180,E1 -9438.523,E2 -9438.523} C_VEL
LIN {X 0,Y 432.173,Z 759.579,A -85,B 0,C 180,E1 -9439.931,E2 -9439.931} C_VEL
LIN {X 0,Y 431.748,Z 766.894,A -85,B 0,C 180,E1 -9441.339,E2 -9441.339} C_VEL
LIN {X 0,Y 431.529,Z 771.838,A -85,B 0,C 180,E1 -9442.512,E2 -9442.512} C_VEL
LIN {X 0,Y 431.295,Z 776.907,A -85,B 0,C 180,E1 -9444.008,E2 -9444.008} C_VEL
LIN {X 0,Y 431.277,Z 780.304,A -85,B 0,C 180,E1 -9445.325,E2 -9445.325} C_VEL
LIN {X 0,Y 431.191,Z 782.196,A -85,B 0,C 180,E1 -9446.261,E2 -9446.261} C_VEL
LIN {X 0,Y 431.237,Z 783.623,A -85,B 0,C 180,E1 -9447.196,E2 -9447.196} C_VEL
LIN {X 0,Y 431.203,Z 784.632,A -85,B 0,C 180,E1 -9448.131,E2 -9448.131} C_VEL
LIN {X 0,Y 431.167,Z 785.471,A -85,B 0,C 180,E1 -9449.999,E2 -9449.999} C_VEL
LIN {X 0,Y 431.169,Z 785.258,A -85,B 0,C 180,E1 -9450.933,E2 -9450.933} C_VEL
LIN {X 0,Y 431.203,Z 784.645,A -85,B 0,C 180,E1 -9451.867,E2 -9451.867} C_VEL
LIN {X 0,Y 431.236,Z 783.638,A -85,B 0,C 180,E1 -9452.801,E2 -9452.801} C_VEL
LIN {X 0,Y 431.19,Z 782.226,A -85,B 0,C 180,E1 -9453.737,E2 -9453.737} C_VEL
LIN {X 0,Y 431.303,Z 779.26,A -85,B 0,C 180,E1 -9455.14,E2 -9455.14} C_VEL
LIN {X 0,Y 431.377,Z 775.245,A -85,B 0,C 180,E1 -9456.547,E2 -9456.547} C_VEL
LIN {X 0,Y 431.636,Z 769.073,A -85,B 0,C 180,E1 -9458.189,E2 -9458.189} C_VEL
LIN {X 0,Y 432.013,Z 762.331,A -85,B 0,C 180,E1 -9459.597,E2 -9459.597} C_VEL
LIN {X 0,Y 432.508,Z 753.97,A -85,B 0,C 180,E1 -9461.006,E2 -9461.006} C_VEL
LIN {X 0,Y 433.133,Z 745.397,A -85,B 0,C 180,E1 -9462.176,E2 -9462.176} C_VEL
LIN {X 0,Y 433.676,Z 735.74,A -85,B 0,C 180,E1 -9463.257,E2 -9463.257} C_VEL
LIN {X 0,Y 434.417,Z 724.354,A -85,B 0,C 180,E1 -9464.282,E2 -9464.282} C_VEL
LIN {X 0,Y 435.012,Z 712.87,A -85,B 0,C 180,E1 -9465.099,E2 -9465.099} C_VEL
LIN {X 0,Y 435.695,Z 699.72,A -85,B 0,C 180,E1 -9465.794,E2 -9465.794} C_VEL
LIN {X 0,Y 436.204,Z 686.494,A -85,B 0,C 180,E1 -9466.285,E2 -9466.285} C_VEL
LIN {X 0,Y 436.564,Z 671.877,A -85,B 0,C 180,E1 -9466.602,E2 -9466.602} C_VEL
LIN {X 0,Y 437.337,Z 595.642,A -85,B 0,C 180,E1 -9467.91,E2 -9467.91} C_VEL
LIN {X 0,Y 433.605,Z 572.692,A -85,B 0,C 180,E1 -9468.489,E2 -9468.489} C_VEL
LIN {X 0,Y 434.631,Z 555.512,A -85,B 0,C 180,E1 -9471.832,E2 -9471.832} C_VEL
LIN {X 0,Y 435.244,Z 545.528,A -85,B 0,C 180,E1 -9473.807,E2 -9473.807} C_VEL
LIN {X 0,Y 433.696,Z 536.798,A -85,B 0,C 180,E1 -9475.687,E2 -9475.687} C_VEL
LIN {X 0,Y 432.421,Z 530.624,A -85,B 0,C 180,E1 -9477.068,E2 -9477.068} C_VEL
LIN {X 0,Y 432.345,Z 530.633,A -85,B 0,C 180,E1 -9480.509,E2 -9480.509} C_VEL
LIN {X 0,Y 432.356,Z 530.628,A -85,B 0,C 180,E1 -9484.002,E2 -9484.002} C_VEL
LIN {X 0,Y 432.33,Z 530.635,A -85,B 0,C 180,E1 -9487.198,E2 -9487.198} C_VEL
LIN {X 0,Y 432.351,Z 530.63,A -85,B 0,C 180,E1 -9490.181,E2 -9490.181} C_VEL
LIN {X 0,Y 432.318,Z 530.636,A -85,B 0,C 180,E1 -9493.059,E2 -9493.059} C_VEL
LIN {X 0,Y 432.327,Z 530.637,A -85,B 0,C 180,E1 -9495.663,E2 -9495.663} C_VEL
LIN {X 0,Y 432.36,Z 530.627,A -85,B 0,C 180,E1 -9498.391,E2 -9498.391} C_VEL
LIN {X 0,Y 432.345,Z 530.628,A -85,B 0,C 180,E1 -9501.85,E2 -9501.85} C_VEL
LIN {X 0,Y 432.333,Z 530.632,A -85,B 0,C 180,E1 -9505.322,E2 -9505.322} C_VEL
LIN {X 0,Y 432.315,Z 530.63,A -85,B 0,C 180,E1 -9508.653,E2 -9508.653} C_VEL
LIN {X 0,Y 432.372,Z 530.63,A -85,B 0,C 180,E1 -9511.368,E2 -9511.368} C_VEL
LIN {X 0,Y 432.355,Z 530.628,A -85,B 0,C 180,E1 -9513.966,E2 -9513.966} C_VEL
LIN {X 0,Y 432.309,Z 530.629,A -85,B 0,C 180,E1 -9517.035,E2 -9517.035} C_VEL
LIN {X 0,Y 432.376,Z 530.617,A -85,B 0,C 180,E1 -9520.514,E2 -9520.514} C_VEL
LIN {X 0,Y 432.42,Z 530.614,A -85,B 0,C 180,E1 -9523.96,E2 -9523.96} C_VEL
LIN {X 0,Y 432.47,Z 530.61,A -85,B 0,C 180,E1 -9527.803,E2 -9527.803} C_VEL
LIN {X 0,Y 432.481,Z 530.611,A -85,B 0,C 180,E1 -9531.59,E2 -9531.59} C_VEL
LIN {X 0,Y 432.588,Z 530.596,A -85,B 0,C 180,E1 -9534.406,E2 -9534.406} C_VEL
LIN {X 0,Y 432.595,Z 530.594,A -85,B 0,C 180,E1 -9538.138,E2 -9538.138} C_VEL
LIN {X 0,Y 432.723,Z 530.582,A -85,B 0,C 180,E1 -9540,E2 -9540} C_VEL
LIN {X 0,Y 432.596,Z 530.596,A -85,B 0,C 180,E1 -9542.793,E2 -9542.793} C_VEL
LIN {X 0,Y 432.564,Z 530.601,A -85,B 0,C 180,E1 -9546.53,E2 -9546.53} C_VEL
LIN {X 0,Y 432.433,Z 530.621,A -85,B 0,C 180,E1 -9549.353,E2 -9549.353} C_VEL
LIN {X 0,Y 432.433,Z 530.619,A -85,B 0,C 180,E1 -9552.812,E2 -9552.812} C_VEL
LIN {X 0,Y 432.4,Z 530.624,A -85,B 0,C 180,E1 -9556.479,E2 -9556.479} C_VEL
LIN {X 0,Y 432.326,Z 530.633,A -85,B 0,C 180,E1 -9559.96,E2 -9559.96} C_VEL
LIN {X 0,Y 432.307,Z 530.637,A -85,B 0,C 180,E1 -9562.964,E2 -9562.964} C_VEL
LIN {X 0,Y 432.35,Z 530.63,A -85,B 0,C 180,E1 -9566.033,E2 -9566.033} C_VEL
LIN {X 0,Y 432.406,Z 530.777,A -85,B 0,C 180,E1 -9566.8,E2 -9566.8} C_VEL
LIN {X 0,Y 434.33,Z 540.735,A -85,B 0,C 180,E1 -9569.305,E2 -9569.305} C_VEL
LIN {X 0,Y 433.915,Z 550.655,A -85,B 0,C 180,E1 -9571.591,E2 -9571.591} C_VEL
LIN {X 0,Y 437.593,Z 569.076,A -85,B 0,C 180,E1 -9572.092,E2 -9572.092} C_VEL
LIN {X 0,Y 436.455,Z 657.468,A -85,B 0,C 180,E1 -9573.625,E2 -9573.625} C_VEL
LIN {X 0,Y 436.08,Z 670.266,A -85,B 0,C 180,E1 -9574.023,E2 -9574.023} C_VEL
LIN {X 0,Y 435.629,Z 682.764,A -85,B 0,C 180,E1 -9574.598,E2 -9574.598} C_VEL
LIN {X 0,Y 435.084,Z 694.296,A -85,B 0,C 180,E1 -9575.313,E2 -9575.313} C_VEL
LIN {X 0,Y 434.4,Z 706.106,A -85,B 0,C 180,E1 -9576.266,E2 -9576.266} C_VEL
LIN {X 0,Y 433.758,Z 716.405,A -85,B 0,C 180,E1 -9577.308,E2 -9577.308} C_VEL
LIN {X 0,Y 433.163,Z 725.414,A -85,B 0,C 180,E1 -9578.427,E2 -9578.427} C_VEL
LIN {X 0,Y 432.582,Z 734.008,A -85,B 0,C 180,E1 -9579.746,E2 -9579.746} C_VEL
LIN {X 0,Y 432.031,Z 742.136,A -85,B 0,C 180,E1 -9581.303,E2 -9581.303} C_VEL
LIN {X 0,Y 431.684,Z 748.602,A -85,B 0,C 180,E1 -9582.896,E2 -9582.896} C_VEL
LIN {X 0,Y 431.426,Z 753.444,A -85,B 0,C 180,E1 -9584.465,E2 -9584.465} C_VEL
LIN {X 0,Y 431.258,Z 756.549,A -85,B 0,C 180,E1 -9585.81,E2 -9585.81} C_VEL
LIN {X 0,Y 431.143,Z 758.788,A -85,B 0,C 180,E1 -9587.183,E2 -9587.183} C_VEL
LIN {X 0,Y 431.052,Z 760.159,A -85,B 0,C 180,E1 -9588.589,E2 -9588.589} C_VEL
LIN {X 0,Y 431.016,Z 760.616,A -85,B 0,C 180,E1 -9590.028,E2 -9590.028} C_VEL
LIN {X 0,Y 431.064,Z 759.92,A -85,B 0,C 180,E1 -9591.719,E2 -9591.719} C_VEL
LIN {X 0,Y 431.099,Z 758.526,A -85,B 0,C 180,E1 -9593.017,E2 -9593.017} C_VEL
LIN {X 0,Y 431.281,Z 755.783,A -85,B 0,C 180,E1 -9594.565,E2 -9594.565} C_VEL
LIN {X 0,Y 431.459,Z 751.635,A -85,B 0,C 180,E1 -9596.173,E2 -9596.173} C_VEL
LIN {X 0,Y 431.796,Z 745.9,A -85,B 0,C 180,E1 -9597.817,E2 -9597.817} C_VEL
LIN {X 0,Y 432.172,Z 738.954,A -85,B 0,C 180,E1 -9599.351,E2 -9599.351} C_VEL
LIN {X 0,Y 432.711,Z 730.372,A -85,B 0,C 180,E1 -9600.842,E2 -9600.842} C_VEL
LIN {X 0,Y 433.285,Z 721.583,A -85,B 0,C 180,E1 -9602.074,E2 -9602.074} C_VEL
LIN {X 0,Y 433.837,Z 712.644,A -85,B 0,C 180,E1 -9603.101,E2 -9603.101} C_VEL
LIN {X 0,Y 434.525,Z 701.774,A -85,B 0,C 180,E1 -9604.108,E2 -9604.108} C_VEL
LIN {X 0,Y 435.101,Z 690.174,A -85,B 0,C 180,E1 -9604.963,E2 -9604.963} C_VEL
LIN {X 0,Y 435.678,Z 677.985,A -85,B 0,C 180,E1 -9605.649,E2 -9605.649} C_VEL
LIN {X 0,Y 436.08,Z 665.147,A -85,B 0,C 180,E1 -9606.163,E2 -9606.163} C_VEL
LIN {X 0,Y 436.374,Z 651.478,A -85,B 0,C 180,E1 -9606.507,E2 -9606.507} C_VEL
LIN {X 0,Y 436.527,Z 636.295,A -85,B 0,C 180,E1 -9606.765,E2 -9606.765} C_VEL
LIN {X 0,Y 435.942,Z 630.49,A -85,B 0,C 180,E1 -9606.889,E2 -9606.889} C_VEL
LIN {X 0,Y 430.72,Z 611.777,A -85,B 0,C 180,E1 -9607.416,E2 -9607.416} C_VEL
LIN {X 0,Y 430.135,Z 605.971,A -85,B 0,C 180,E1 -9607.542,E2 -9607.542} C_VEL
LIN {X 0,Y 430.447,Z 568.733,A -85,B 0,C 180,E1 -9608.197,E2 -9608.197} C_VEL
LIN {X 0,Y 426.796,Z 550.135,A -85,B 0,C 180,E1 -9608.699,E2 -9608.699} C_VEL
LIN {X 0,Y 427.18,Z 542.152,A -85,B 0,C 180,E1 -9610.541,E2 -9610.541} C_VEL
LIN {X 0,Y 425.41,Z 531.496,A -85,B 0,C 180,E1 -9613.181,E2 -9613.181} C_VEL
LIN {X 0,Y 425.389,Z 531.499,A -85,B 0,C 180,E1 -9617.097,E2 -9617.097} C_VEL
LIN {X 0,Y 425.397,Z 531.495,A -85,B 0,C 180,E1 -9620.492,E2 -9620.492} C_VEL
LIN {X 0,Y 425.519,Z 531.478,A -85,B 0,C 180,E1 -9623.362,E2 -9623.362} C_VEL
LIN {X 0,Y 425.367,Z 531.498,A -85,B 0,C 180,E1 -9625.263,E2 -9625.263} C_VEL
LIN {X 0,Y 425.573,Z 531.469,A -85,B 0,C 180,E1 -9628.109,E2 -9628.109} C_VEL
LIN {X 0,Y 425.701,Z 531.453,A -85,B 0,C 180,E1 -9630.001,E2 -9630.001} C_VEL
LIN {X 0,Y 425.554,Z 531.478,A -85,B 0,C 180,E1 -9632.841,E2 -9632.841} C_VEL
LIN {X 0,Y 425.521,Z 531.479,A -85,B 0,C 180,E1 -9636.64,E2 -9636.64} C_VEL
LIN {X 0,Y 425.399,Z 531.493,A -85,B 0,C 180,E1 -9639.511,E2 -9639.511} C_VEL
LIN {X 0,Y 425.392,Z 531.498,A -85,B 0,C 180,E1 -9642.905,E2 -9642.905} C_VEL
LIN {X 0,Y 425.36,Z 531.498,A -85,B 0,C 180,E1 -9646.606,E2 -9646.606} C_VEL
LIN {X 0,Y 425.328,Z 531.502,A -85,B 0,C 180,E1 -9649.637,E2 -9649.637} C_VEL
LIN {X 0,Y 425.307,Z 531.507,A -85,B 0,C 180,E1 -9653.366,E2 -9653.366} C_VEL
LIN {X 0,Y 425.348,Z 531.501,A -85,B 0,C 180,E1 -9656.845,E2 -9656.845} C_VEL
LIN {X 0,Y 425.292,Z 531.506,A -85,B 0,C 180,E1 -9659.721,E2 -9659.721} C_VEL
LIN {X 0,Y 425.283,Z 531.51,A -85,B 0,C 180,E1 -9663.049,E2 -9663.049} C_VEL
LIN {X 0,Y 425.284,Z 531.506,A -85,B 0,C 180,E1 -9665.93,E2 -9665.93} C_VEL
LIN {X 0,Y 425.299,Z 531.508,A -85,B 0,C 180,E1 -9669.045,E2 -9669.045} C_VEL
LIN {X 0,Y 425.281,Z 531.506,A -85,B 0,C 180,E1 -9672.654,E2 -9672.654} C_VEL
LIN {X 0,Y 425.264,Z 531.508,A -85,B 0,C 180,E1 -9676.045,E2 -9676.045} C_VEL
LIN {X 0,Y 425.277,Z 531.506,A -85,B 0,C 180,E1 -9678.622,E2 -9678.622} C_VEL
LIN {X 0,Y 425.309,Z 531.506,A -85,B 0,C 180,E1 -9681.103,E2 -9681.103} C_VEL
LIN {X 0,Y 425.303,Z 531.503,A -85,B 0,C 180,E1 -9684.665,E2 -9684.665} C_VEL
LIN {X 0,Y 425.269,Z 531.508,A -85,B 0,C 180,E1 -9688.074,E2 -9688.074} C_VEL
LIN {X 0,Y 425.336,Z 531.504,A -85,B 0,C 180,E1 -9691.369,E2 -9691.369} C_VEL
LIN {X 0,Y 425.297,Z 531.503,A -85,B 0,C 180,E1 -9694.555,E2 -9694.555} C_VEL
LIN {X 0,Y 425.293,Z 531.511,A -85,B 0,C 180,E1 -9697.662,E2 -9697.662} C_VEL
LIN {X 0,Y 425.367,Z 531.495,A -85,B 0,C 180,E1 -9700.705,E2 -9700.705} C_VEL
LIN {X 0,Y 425.394,Z 531.499,A -85,B 0,C 180,E1 -9703.689,E2 -9703.689} C_VEL
LIN {X 0,Y 425.418,Z 531.495,A -85,B 0,C 180,E1 -9707.599,E2 -9707.599} C_VEL
LIN {X 0,Y 425.449,Z 531.489,A -85,B 0,C 180,E1 -9711.451,E2 -9711.451} C_VEL
LIN {X 0,Y 425.558,Z 531.473,A -85,B 0,C 180,E1 -9714.314,E2 -9714.314} C_VEL
LIN {X 0,Y 425.58,Z 531.472,A -85,B 0,C 180,E1 -9718.108,E2 -9718.108} C_VEL
LIN {X 0,Y 425.708,Z 531.458,A -85,B 0,C 180,E1 -9720,E2 -9720} C_VEL
LIN {X 0,Y 425.552,Z 531.472,A -85,B 0,C 180,E1 -9722.84,E2 -9722.84} C_VEL
LIN {X 0,Y 425.539,Z 531.474,A -85,B 0,C 180,E1 -9726.639,E2 -9726.639} C_VEL
LIN {X 0,Y 425.407,Z 531.493,A -85,B 0,C 180,E1 -9729.51,E2 -9729.51} C_VEL
LIN {X 0,Y 425.401,Z 531.49,A -85,B 0,C 180,E1 -9732.904,E2 -9732.904} C_VEL
LIN {X 0,Y 425.369,Z 531.496,A -85,B 0,C 180,E1 -9736.605,E2 -9736.605} C_VEL
LIN {X 0,Y 425.336,Z 531.502,A -85,B 0,C 180,E1 -9739.636,E2 -9739.636} C_VEL
LIN {X 0,Y 425.296,Z 531.508,A -85,B 0,C 180,E1 -9742.339,E2 -9742.339} C_VEL
LIN {X 0,Y 425.299,Z 531.504,A -85,B 0,C 180,E1 -9745.446,E2 -9745.446} C_VEL
LIN {X 0,Y 425.357,Z 531.498,A -85,B 0,C 180,E1 -9747.558,E2 -9747.558} C_VEL
LIN {X 0,Y 425.296,Z 531.505,A -85,B 0,C 180,E1 -9750.816,E2 -9750.816} C_VEL
LIN {X 0,Y 425.319,Z 531.507,A -85,B 0,C 180,E1 -9754.288,E2 -9754.288} C_VEL
LIN {X 0,Y 425.285,Z 531.507,A -85,B 0,C 180,E1 -9757.694,E2 -9757.694} C_VEL
LIN {X 0,Y 425.284,Z 531.509,A -85,B 0,C 180,E1 -9760.519,E2 -9760.519} C_VEL
LIN {X 0,Y 425.268,Z 531.511,A -85,B 0,C 180,E1 -9763.956,E2 -9763.956} C_VEL
LIN {X 0,Y 425.282,Z 531.505,A -85,B 0,C 180,E1 -9767.346,E2 -9767.346} C_VEL
LIN {X 0,Y 425.311,Z 531.503,A -85,B 0,C 180,E1 -9770.955,E2 -9770.955} C_VEL
LIN {X 0,Y 425.306,Z 531.507,A -85,B 0,C 180,E1 -9774.663,E2 -9774.663} C_VEL
LIN {X 0,Y 425.272,Z 531.51,A -85,B 0,C 180,E1 -9778.072,E2 -9778.072} C_VEL
LIN {X 0,Y 425.338,Z 531.501,A -85,B 0,C 180,E1 -9781.367,E2 -9781.367} C_VEL
LIN {X 0,Y 425.398,Z 531.57,A -85,B 0,C 180,E1 -9782.837,E2 -9782.837} C_VEL
LIN {X 0,Y 427.759,Z 543.742,A -85,B 0,C 180,E1 -9785.497,E2 -9785.497} C_VEL
LIN {X 0,Y 428.215,Z 547.51,A -85,B 0,C 180,E1 -9786.289,E2 -9786.289} C_VEL
LIN {X 0,Y 427.246,Z 562.625,A -85,B 0,C 180,E1 -9789.288,E2 -9789.288} C_VEL
LIN {X 0,Y 426.655,Z 573.015,A -85,B 0,C 180,E1 -9791.326,E2 -9791.326} C_VEL
LIN {X 0,Y 430.358,Z 597.415,A -85,B 0,C 180,E1 -9791.923,E2 -9791.923} C_VEL
LIN {X 0,Y 429.379,Z 682.052,A -85,B 0,C 180,E1 -9793.415,E2 -9793.415} C_VEL
LIN {X 0,Y 428.851,Z 695.673,A -85,B 0,C 180,E1 -9793.853,E2 -9793.853} C_VEL
LIN {X 0,Y 428.278,Z 708.5,A -85,B 0,C 180,E1 -9794.472,E2 -9794.472} C_VEL
LIN {X 0,Y 427.619,Z 720.248,A -85,B 0,C 180,E1 -9795.24,E2 -9795.24} C_VEL
LIN {X 0,Y 426.974,Z 730.978,A -85,B 0,C 180,E1 -9796.133,E2 -9796.133} C_VEL
LIN {X 0,Y 426.31,Z 741.828,A -85,B 0,C 180,E1 -9797.261,E2 -9797.261} C_VEL
LIN {X 0,Y 425.603,Z 751.846,A -85,B 0,C 180,E1 -9798.57,E2 -9798.57} C_VEL
LIN {X 0,Y 425.061,Z 760.668,A -85,B 0,C 180,E1 -9800.001,E2 -9800.001} C_VEL
LIN {X 0,Y 424.653,Z 767.702,A -85,B 0,C 180,E1 -9801.433,E2 -9801.433} C_VEL
LIN {X 0,Y 424.361,Z 773.328,A -85,B 0,C 180,E1 -9802.864,E2 -9802.864} C_VEL
LIN {X 0,Y 424.203,Z 777.745,A -85,B 0,C 180,E1 -9804.294,E2 -9804.294} C_VEL
LIN {X 0,Y 424.206,Z 780.078,A -85,B 0,C 180,E1 -9805.247,E2 -9805.247} C_VEL
LIN {X 0,Y 424.102,Z 781.974,A -85,B 0,C 180,E1 -9806.198,E2 -9806.198} C_VEL
LIN {X 0,Y 424.133,Z 783.408,A -85,B 0,C 180,E1 -9807.149,E2 -9807.149} C_VEL
LIN {X 0,Y 424.129,Z 784.421,A -85,B 0,C 180,E1 -9808.099,E2 -9808.099} C_VEL
LIN {X 0,Y 424.084,Z 785.266,A -85,B 0,C 180,E1 -9809.999,E2 -9809.999} C_VEL
LIN {X 0,Y 424.088,Z 785.057,A -85,B 0,C 180,E1 -9810.948,E2 -9810.948} C_VEL
LIN {X 0,Y 424.129,Z 784.444,A -85,B 0,C 180,E1 -9811.898,E2 -9811.898} C_VEL
LIN {X 0,Y 424.132,Z 783.438,A -85,B 0,C 180,E1 -9812.848,E2 -9812.848} C_VEL
LIN {X 0,Y 424.101,Z 782.028,A -85,B 0,C 180,E1 -9813.799,E2 -9813.799} C_VEL
LIN {X 0,Y 424.216,Z 779.063,A -85,B 0,C 180,E1 -9815.227,E2 -9815.227} C_VEL
LIN {X 0,Y 424.301,Z 775.052,A -85,B 0,C 180,E1 -9816.657,E2 -9816.657} C_VEL
LIN {X 0,Y 424.59,Z 768.889,A -85,B 0,C 180,E1 -9818.326,E2 -9818.326} C_VEL
LIN {X 0,Y 424.982,Z 762.157,A -85,B 0,C 180,E1 -9819.758,E2 -9819.758} C_VEL
LIN {X 0,Y 425.496,Z 753.809,A -85,B 0,C 180,E1 -9821.189,E2 -9821.189} C_VEL
LIN {X 0,Y 426.181,Z 745.251,A -85,B 0,C 180,E1 -9822.378,E2 -9822.378} C_VEL
LIN {X 0,Y 426.806,Z 734.944,A -85,B 0,C 180,E1 -9823.542,E2 -9823.542} C_VEL
LIN {X 0,Y 427.519,Z 724.232,A -85,B 0,C 180,E1 -9824.517,E2 -9824.517} C_VEL
LIN {X 0,Y 428.168,Z 712.775,A -85,B 0,C 180,E1 -9825.346,E2 -9825.346} C_VEL
LIN {X 0,Y 428.868,Z 699.676,A -85,B 0,C 180,E1 -9826.052,E2 -9826.052} C_VEL
LIN {X 0,Y 429.401,Z 686.527,A -85,B 0,C 180,E1 -9826.551,E2 -9826.551} C_VEL
LIN {X 0,Y 429.748,Z 673.892,A -85,B 0,C 180,E1 -9826.843,E2 -9826.843} C_VEL
LIN {X 0,Y 430.51,Z 595.628,A -85,B 0,C 180,E1 -9828.213,E2 -9828.213} C_VEL
LIN {X 0,Y 426.702,Z 572.457,A -85,B 0,C 180,E1 -9828.82,E2 -9828.82} C_VEL
LIN {X 0,Y 427.875,Z 554.186,A -85,B 0,C 180,E1 -9832.445,E2 -9832.445} C_VEL
LIN {X 0,Y 428.313,Z 546.693,A -85,B 0,C 180,E1 -9833.959,E2 -9833.959} C_VEL
LIN {X 0,Y 426.234,Z 535.514,A -85,B 0,C 180,E1 -9836.434,E2 -9836.434} C_VEL
LIN {X 0,Y 425.352,Z 531.505,A -85,B 0,C 180,E1 -9837.368,E2 -9837.368} C_VEL
LIN {X 0,Y 425.285,Z 531.511,A -85,B 0,C 180,E1 -9840.814,E2 -9840.814} C_VEL
LIN {X 0,Y 425.308,Z 531.505,A -85,B 0,C 180,E1 -9844.286,E2 -9844.286} C_VEL
LIN {X 0,Y 425.284,Z 531.515,A -85,B 0,C 180,E1 -9847.692,E2 -9847.692} C_VEL
LIN {X 0,Y 425.295,Z 531.508,A -85,B 0,C 180,E1 -9850.522,E2 -9850.522} C_VEL
LIN {X 0,Y 425.258,Z 531.518,A -85,B 0,C 180,E1 -9853.35,E2 -9853.35} C_VEL
LIN {X 0,Y 425.251,Z 531.513,A -85,B 0,C 180,E1 -9856.648,E2 -9856.648} C_VEL
LIN {X 0,Y 425.292,Z 531.509,A -85,B 0,C 180,E1 -9859.475,E2 -9859.475} C_VEL
LIN {X 0,Y 425.279,Z 531.505,A -85,B 0,C 180,E1 -9862.486,E2 -9862.486} C_VEL
LIN {X 0,Y 425.3,Z 531.505,A -85,B 0,C 180,E1 -9865.816,E2 -9865.816} C_VEL
LIN {X 0,Y 425.292,Z 531.507,A -85,B 0,C 180,E1 -9869.235,E2 -9869.235} C_VEL
LIN {X 0,Y 425.341,Z 531.496,A -85,B 0,C 180,E1 -9872.441,E2 -9872.441} C_VEL
LIN {X 0,Y 425.342,Z 531.5,A -85,B 0,C 180,E1 -9875.601,E2 -9875.601} C_VEL
LIN {X 0,Y 425.283,Z 531.507,A -85,B 0,C 180,E1 -9878.681,E2 -9878.681} C_VEL
LIN {X 0,Y 425.323,Z 531.506,A -85,B 0,C 180,E1 -9881.702,E2 -9881.702} C_VEL
LIN {X 0,Y 425.338,Z 531.495,A -85,B 0,C 180,E1 -9884.67,E2 -9884.67} C_VEL
LIN {X 0,Y 425.419,Z 531.49,A -85,B 0,C 180,E1 -9887.598,E2 -9887.598} C_VEL
LIN {X 0,Y 425.432,Z 531.489,A -85,B 0,C 180,E1 -9891.449,E2 -9891.449} C_VEL
LIN {X 0,Y 425.544,Z 531.474,A -85,B 0,C 180,E1 -9894.313,E2 -9894.313} C_VEL
LIN {X 0,Y 425.564,Z 531.47,A -85,B 0,C 180,E1 -9898.107,E2 -9898.107} C_VEL
LIN {X 0,Y 425.693,Z 531.458,A -85,B 0,C 180,E1 -9900,E2 -9900} C_VEL
LIN {X 0,Y 425.548,Z 531.474,A -85,B 0,C 180,E1 -9902.839,E2 -9902.839} C_VEL
LIN {X 0,Y 425.567,Z 531.476,A -85,B 0,C 180,E1 -9905.686,E2 -9905.686} C_VEL
LIN {X 0,Y 425.431,Z 531.489,A -85,B 0,C 180,E1 -9908.55,E2 -9908.55} C_VEL
LIN {X 0,Y 425.42,Z 531.491,A -85,B 0,C 180,E1 -9912.401,E2 -9912.401} C_VEL
LIN {X 0,Y 425.376,Z 531.499,A -85,B 0,C 180,E1 -9916.312,E2 -9916.312} C_VEL
LIN {X 0,Y 425.316,Z 531.508,A -85,B 0,C 180,E1 -9919.636,E2 -9919.636} C_VEL
LIN {X 0,Y 425.294,Z 531.509,A -85,B 0,C 180,E1 -9923.365,E2 -9923.365} C_VEL
LIN {X 0,Y 425.356,Z 531.537,A -85,B 0,C 180,E1 -9926.494,E2 -9926.494} C_VEL
LIN {X 0,Y 427.245,Z 541.041,A -85,B 0,C 180,E1 -9928.942,E2 -9928.942} C_VEL
LIN {X 0,Y 427.338,Z 545.864,A -85,B 0,C 180,E1 -9930.105,E2 -9930.105} C_VEL
LIN {X 0,Y 427.023,Z 550.734,A -85,B 0,C 180,E1 -9931.247,E2 -9931.247} C_VEL
LIN {X 0,Y 430.8,Z 569.124,A -85,B 0,C 180,E1 -9931.781,E2 -9931.781} C_VEL
LIN {X 0,Y 429.683,Z 657.655,A -85,B 0,C 180,E1 -9933.35,E2 -9933.35} C_VEL
LIN {X 0,Y 429.285,Z 670.802,A -85,B 0,C 180,E1 -9933.767,E2 -9933.767} C_VEL
LIN {X 0,Y 428.787,Z 683.449,A -85,B 0,C 180,E1 -9934.363,E2 -9934.363} C_VEL
LIN {X 0,Y 428.184,Z 695.438,A -85,B 0,C 180,E1 -9935.134,E2 -9935.134} C_VEL
LIN {X 0,Y 427.462,Z 707.134,A -85,B 0,C 180,E1 -9936.106,E2 -9936.106} C_VEL
LIN {X 0,Y 426.718,Z 718,A -85,B 0,C 180,E1 -9937.247,E2 -9937.247} C_VEL
LIN {X 0,Y 426.073,Z 727.707,A -85,B 0,C 180,E1 -9938.53,E2 -9938.53} C_VEL
LIN {X 0,Y 425.487,Z 735.813,A -85,B 0,C 180,E1 -9939.847,E2 -9939.847} C_VEL
LIN {X 0,Y 424.938,Z 743.543,A -85,B 0,C 180,E1 -9941.418,E2 -9941.418} C_VEL
LIN {X 0,Y 424.653,Z 748.682,A -85,B 0,C 180,E1 -9942.73,E2 -9942.73} C_VEL
LIN {X 0,Y 424.421,Z 752.875,A -85,B 0,C 180,E1 -9944.065,E2 -9944.065} C_VEL
LIN {X 0,Y 424.152,Z 757.076,A -85,B 0,C 180,E1 -9945.902,E2 -9945.902} C_VEL
LIN {X 0,Y 424.045,Z 759.076,A -85,B 0,C 180,E1 -9947.196,E2 -9947.196} C_VEL
LIN {X 0,Y 423.96,Z 760.311,A -85,B 0,C 180,E1 -9948.467,E2 -9948.467} C_VEL
LIN {X 0,Y 423.928,Z 760.782,A -85,B 0,C 180,E1 -9949.72,E2 -9949.72} C_VEL
LIN {X 0,Y 423.925,Z 760.479,A -85,B 0,C 180,E1 -9951.185,E2 -9951.185} C_VEL
LIN {X 0,Y 423.994,Z 759.147,A -85,B 0,C 180,E1 -9952.714,E2 -9952.714} C_VEL
LIN {X 0,Y 424.199,Z 756.138,A -85,B 0,C 180,E1 -9954.561,E2 -9954.561} C_VEL
LIN {X 0,Y 424.428,Z 751.444,A -85,B 0,C 180,E1 -9956.394,E2 -9956.394} C_VEL
LIN {X 0,Y 424.754,Z 745.729,A -85,B 0,C 180,E1 -9958.032,E2 -9958.032} C_VEL
LIN {X 0,Y 425.166,Z 738.895,A -85,B 0,C 180,E1 -9959.542,E2 -9959.542} C_VEL
LIN {X 0,Y 425.734,Z 730.392,A -85,B 0,C 180,E1 -9961.034,E2 -9961.034} C_VEL
LIN {X 0,Y 426.36,Z 720.793,A -85,B 0,C 180,E1 -9962.382,E2 -9962.382} C_VEL
LIN {X 0,Y 426.976,Z 710.943,A -85,B 0,C 180,E1 -9963.493,E2 -9963.493} C_VEL
LIN {X 0,Y 427.673,Z 700.475,A -85,B 0,C 180,E1 -9964.448,E2 -9964.448} C_VEL
LIN {X 0,Y 428.279,Z 688.25,A -85,B 0,C 180,E1 -9965.33,E2 -9965.33} C_VEL
LIN {X 0,Y 428.879,Z 675.801,A -85,B 0,C 180,E1 -9965.996,E2 -9965.996} C_VEL
LIN {X 0,Y 429.365,Z 662.76,A -85,B 0,C 180,E1 -9966.49,E2 -9966.49} C_VEL
LIN {X 0,Y 429.611,Z 649.259,A -85,B 0,C 180,E1 -9966.799,E2 -9966.799} C_VEL
LIN {X 0,Y 430.135,Z 605.971,A -85,B 0,C 180,E1 -9967.542,E2 -9967.542} C_VEL
LIN {X 0,Y 429.543,Z 600.166,A -85,B 0,C 180,E1 -9967.669,E2 -9967.669} C_VEL
LIN {X 0,Y 424.291,Z 581.478,A -85,B 0,C 180,E1 -9968.224,E2 -9968.224} C_VEL
LIN {X 0,Y 423.711,Z 575.673,A -85,B 0,C 180,E1 -9968.355,E2 -9968.355} C_VEL
LIN {X 0,Y 423.535,Z 568.997,A -85,B 0,C 180,E1 -9968.485,E2 -9968.485} C_VEL
LIN {X 0,Y 419.852,Z 550.299,A -85,B 0,C 180,E1 -9969.005,E2 -9969.005} C_VEL
LIN {X 0,Y 420.185,Z 543.034,A -85,B 0,C 180,E1 -9970.712,E2 -9970.712} C_VEL
LIN {X 0,Y 418.352,Z 532.376,A -85,B 0,C 180,E1 -9973.408,E2 -9973.408} C_VEL
LIN {X 0,Y 418.341,Z 532.377,A -85,B 0,C 180,E1 -9977,E2 -9977} C_VEL
LIN {X 0,Y 418.337,Z 532.373,A -85,B 0,C 180,E1 -9980.33,E2 -9980.33} C_VEL
LIN {X 0,Y 418.483,Z 532.355,A -85,B 0,C 180,E1 -9983.25,E2 -9983.25} C_VEL
LIN {X 0,Y 418.337,Z 532.374,A -85,B 0,C 180,E1 -9985.183,E2 -9985.183} C_VEL
LIN {X 0,Y 418.542,Z 532.345,A -85,B 0,C 180,E1 -9988.077,E2 -9988.077} C_VEL
LIN {X 0,Y 418.67,Z 532.329,A -85,B 0,C 180,E1 -9990.001,E2 -9990.001} C_VEL
LIN {X 0,Y 418.508,Z 532.356,A -85,B 0,C 180,E1 -9992.889,E2 -9992.889} C_VEL
LIN {X 0,Y 418.485,Z 532.357,A -85,B 0,C 180,E1 -9996.752,E2 -9996.752} C_VEL
LIN {X 0,Y 418.34,Z 532.371,A -85,B 0,C 180,E1 -9999.673,E2 -9999.673} C_VEL
LIN {X 0,Y 418.345,Z 532.377,A -85,B 0,C 180,E1 -10003.002,E2 -10003.002} C_VEL
LIN {X 0,Y 418.312,Z 532.377,A -85,B 0,C 180,E1 -10006.737,E2 -10006.737} C_VEL
LIN {X 0,Y 418.27,Z 532.38,A -85,B 0,C 180,E1 -10009.791,E2 -10009.791} C_VEL
LIN {X 0,Y 418.238,Z 532.386,A -85,B 0,C 180,E1 -10012.737,E2 -10012.737} C_VEL
LIN {X 0,Y 418.271,Z 532.379,A -85,B 0,C 180,E1 -10015.905,E2 -10015.905} C_VEL
LIN {X 0,Y 418.266,Z 532.387,A -85,B 0,C 180,E1 -10019.163,E2 -10019.163} C_VEL
LIN {X 0,Y 418.259,Z 532.383,A -85,B 0,C 180,E1 -10022.845,E2 -10022.845} C_VEL
LIN {X 0,Y 418.246,Z 532.382,A -85,B 0,C 180,E1 -10026.239,E2 -10026.239} C_VEL
LIN {X 0,Y 418.253,Z 532.384,A -85,B 0,C 180,E1 -10029.683,E2 -10029.683} C_VEL
LIN {X 0,Y 418.235,Z 532.383,A -85,B 0,C 180,E1 -10032.323,E2 -10032.323} C_VEL
LIN {X 0,Y 418.241,Z 532.387,A -85,B 0,C 180,E1 -10035.11,E2 -10035.11} C_VEL
LIN {X 0,Y 418.243,Z 532.385,A -85,B 0,C 180,E1 -10037.768,E2 -10037.768} C_VEL
LIN {X 0,Y 418.256,Z 532.381,A -85,B 0,C 180,E1 -10040.621,E2 -10040.621} C_VEL
LIN {X 0,Y 418.247,Z 532.384,A -85,B 0,C 180,E1 -10043.977,E2 -10043.977} C_VEL
LIN {X 0,Y 418.262,Z 532.383,A -85,B 0,C 180,E1 -10047.157,E2 -10047.157} C_VEL
LIN {X 0,Y 418.273,Z 532.38,A -85,B 0,C 180,E1 -10050.896,E2 -10050.896} C_VEL
LIN {X 0,Y 418.274,Z 532.38,A -85,B 0,C 180,E1 -10054.097,E2 -10054.097} C_VEL
LIN {X 0,Y 418.237,Z 532.386,A -85,B 0,C 180,E1 -10057.264,E2 -10057.264} C_VEL
LIN {X 0,Y 418.288,Z 532.377,A -85,B 0,C 180,E1 -10060.365,E2 -10060.365} C_VEL
LIN {X 0,Y 418.322,Z 532.377,A -85,B 0,C 180,E1 -10063.405,E2 -10063.405} C_VEL
LIN {X 0,Y 418.353,Z 532.369,A -85,B 0,C 180,E1 -10067,E2 -10067} C_VEL
LIN {X 0,Y 418.346,Z 532.371,A -85,B 0,C 180,E1 -10070.329,E2 -10070.329} C_VEL
LIN {X 0,Y 418.495,Z 532.353,A -85,B 0,C 180,E1 -10073.25,E2 -10073.25} C_VEL
LIN {X 0,Y 418.344,Z 532.371,A -85,B 0,C 180,E1 -10075.182,E2 -10075.182} C_VEL
LIN {X 0,Y 418.549,Z 532.348,A -85,B 0,C 180,E1 -10078.076,E2 -10078.076} C_VEL
LIN {X 0,Y 418.678,Z 532.334,A -85,B 0,C 180,E1 -10080,E2 -10080} C_VEL
LIN {X 0,Y 418.508,Z 532.349,A -85,B 0,C 180,E1 -10082.888,E2 -10082.888} C_VEL
LIN {X 0,Y 418.501,Z 532.35,A -85,B 0,C 180,E1 -10086.751,E2 -10086.751} C_VEL
LIN {X 0,Y 418.408,Z 532.362,A -85,B 0,C 180,E1 -10088.695,E2 -10088.695} C_VEL
LIN {X 0,Y 418.363,Z 532.368,A -85,B 0,C 180,E1 -10092.615,E2 -10092.615} C_VEL
LIN {X 0,Y 418.31,Z 532.377,A -85,B 0,C 180,E1 -10095.594,E2 -10095.594} C_VEL
LIN {X 0,Y 418.289,Z 532.378,A -85,B 0,C 180,E1 -10098.617,E2 -10098.617} C_VEL
LIN {X 0,Y 418.242,Z 532.386,A -85,B 0,C 180,E1 -10101.696,E2 -10101.696} C_VEL
LIN {X 0,Y 418.292,Z 532.376,A -85,B 0,C 180,E1 -10104.864,E2 -10104.864} C_VEL
LIN {X 0,Y 418.299,Z 532.383,A -85,B 0,C 180,E1 -10108.063,E2 -10108.063} C_VEL
LIN {X 0,Y 418.219,Z 532.386,A -85,B 0,C 180,E1 -10111.396,E2 -10111.396} C_VEL
LIN {X 0,Y 418.273,Z 532.381,A -85,B 0,C 180,E1 -10114.58,E2 -10114.58} C_VEL
LIN {X 0,Y 418.233,Z 532.387,A -85,B 0,C 180,E1 -10117.833,E2 -10117.833} C_VEL
LIN {X 0,Y 418.227,Z 532.385,A -85,B 0,C 180,E1 -10120.948,E2 -10120.948} C_VEL
LIN {X 0,Y 418.215,Z 532.387,A -85,B 0,C 180,E1 -10123.729,E2 -10123.729} C_VEL
LIN {X 0,Y 418.217,Z 532.391,A -85,B 0,C 180,E1 -10126.448,E2 -10126.448} C_VEL
LIN {X 0,Y 418.232,Z 532.384,A -85,B 0,C 180,E1 -10129.129,E2 -10129.129} C_VEL
LIN {X 0,Y 418.241,Z 532.388,A -85,B 0,C 180,E1 -10132.165,E2 -10132.165} C_VEL
LIN {X 0,Y 418.273,Z 532.379,A -85,B 0,C 180,E1 -10135.419,E2 -10135.419} C_VEL
LIN {X 0,Y 418.219,Z 532.392,A -85,B 0,C 180,E1 -10138.603,E2 -10138.603} C_VEL
LIN {X 0,Y 418.305,Z 532.379,A -85,B 0,C 180,E1 -10141.936,E2 -10141.936} C_VEL
LIN {X 0,Y 418.358,Z 532.491,A -85,B 0,C 180,E1 -10142.599,E2 -10142.599} C_VEL
LIN {X 0,Y 420.74,Z 544.699,A -85,B 0,C 180,E1 -10145.316,E2 -10145.316} C_VEL
LIN {X 0,Y 421.277,Z 548.508,A -85,B 0,C 180,E1 -10146.136,E2 -10146.136} C_VEL
LIN {X 0,Y 420.273,Z 563.615,A -85,B 0,C 180,E1 -10149.184,E2 -10149.184} C_VEL
LIN {X 0,Y 419.704,Z 572.816,A -85,B 0,C 180,E1 -10151.019,E2 -10151.019} C_VEL
LIN {X 0,Y 423.575,Z 597.887,A -85,B 0,C 180,E1 -10151.653,E2 -10151.653} C_VEL
LIN {X 0,Y 422.542,Z 681.101,A -85,B 0,C 180,E1 -10153.139,E2 -10153.139} C_VEL
LIN {X 0,Y 422.037,Z 694.965,A -85,B 0,C 180,E1 -10153.585,E2 -10153.585} C_VEL
LIN {X 0,Y 421.494,Z 706.888,A -85,B 0,C 180,E1 -10154.154,E2 -10154.154} C_VEL
LIN {X 0,Y 420.856,Z 718.191,A -85,B 0,C 180,E1 -10154.874,E2 -10154.874} C_VEL
LIN {X 0,Y 420.115,Z 729.484,A -85,B 0,C 180,E1 -10155.8,E2 -10155.8} C_VEL
LIN {X 0,Y 419.369,Z 740.398,A -85,B 0,C 180,E1 -10156.923,E2 -10156.923} C_VEL
LIN {X 0,Y 418.758,Z 749.872,A -85,B 0,C 180,E1 -10158.135,E2 -10158.135} C_VEL
LIN {X 0,Y 418.09,Z 758.998,A -85,B 0,C 180,E1 -10159.588,E2 -10159.588} C_VEL
LIN {X 0,Y 417.664,Z 766.354,A -85,B 0,C 180,E1 -10161.044,E2 -10161.044} C_VEL
LIN {X 0,Y 417.381,Z 771.327,A -85,B 0,C 180,E1 -10162.257,E2 -10162.257} C_VEL
LIN {X 0,Y 417.174,Z 776.116,A -85,B 0,C 180,E1 -10163.7,E2 -10163.7} C_VEL
LIN {X 0,Y 417.114,Z 779.845,A -85,B 0,C 180,E1 -10165.166,E2 -10165.166} C_VEL
LIN {X 0,Y 417.018,Z 781.747,A -85,B 0,C 180,E1 -10166.133,E2 -10166.133} C_VEL
LIN {X 0,Y 417.03,Z 783.189,A -85,B 0,C 180,E1 -10167.101,E2 -10167.101} C_VEL
LIN {X 0,Y 417.057,Z 784.207,A -85,B 0,C 180,E1 -10168.067,E2 -10168.067} C_VEL
LIN {X 0,Y 417.004,Z 785.06,A -85,B 0,C 180,E1 -10169.999,E2 -10169.999} C_VEL
LIN {X 0,Y 417.011,Z 784.857,A -85,B 0,C 180,E1 -10170.964,E2 -10170.964} C_VEL
LIN {X 0,Y 417.056,Z 784.247,A -85,B 0,C 180,E1 -10171.93,E2 -10171.93} C_VEL
LIN {X 0,Y 417.029,Z 783.243,A -85,B 0,C 180,E1 -10172.897,E2 -10172.897} C_VEL
LIN {X 0,Y 417.017,Z 781.838,A -85,B 0,C 180,E1 -10173.864,E2 -10173.864} C_VEL
LIN {X 0,Y 417.131,Z 778.879,A -85,B 0,C 180,E1 -10175.316,E2 -10175.316} C_VEL
LIN {X 0,Y 417.234,Z 774.873,A -85,B 0,C 180,E1 -10176.77,E2 -10176.77} C_VEL
LIN {X 0,Y 417.53,Z 768.72,A -85,B 0,C 180,E1 -10178.468,E2 -10178.468} C_VEL
LIN {X 0,Y 417.945,Z 761.993,A -85,B 0,C 180,E1 -10179.924,E2 -10179.924} C_VEL
LIN {X 0,Y 418.509,Z 753.65,A -85,B 0,C 180,E1 -10181.379,E2 -10181.379} C_VEL
LIN {X 0,Y 419.218,Z 745.103,A -85,B 0,C 180,E1 -10182.586,E2 -10182.586} C_VEL
LIN {X 0,Y 419.906,Z 734.426,A -85,B 0,C 180,E1 -10183.809,E2 -10183.809} C_VEL
LIN {X 0,Y 420.704,Z 722.674,A -85,B 0,C 180,E1 -10184.881,E2 -10184.881} C_VEL
LIN {X 0,Y 421.429,Z 710.729,A -85,B 0,C 180,E1 -10185.722,E2 -10185.722} C_VEL
LIN {X 0,Y 422.128,Z 698.338,A -85,B 0,C 180,E1 -10186.378,E2 -10186.378} C_VEL
LIN {X 0,Y 422.703,Z 685.657,A -85,B 0,C 180,E1 -10186.852,E2 -10186.852} C_VEL
LIN {X 0,Y 423.055,Z 670.816,A -85,B 0,C 180,E1 -10187.179,E2 -10187.179} C_VEL
LIN {X 0,Y 423.868,Z 596.954,A -85,B 0,C 180,E1 -10188.499,E2 -10188.499} C_VEL
LIN {X 0,Y 419.785,Z 572.168,A -85,B 0,C 180,E1 -10189.177,E2 -10189.177} C_VEL
LIN {X 0,Y 421.041,Z 554.301,A -85,B 0,C 180,E1 -10192.789,E2 -10192.789} C_VEL
LIN {X 0,Y 421.373,Z 547.875,A -85,B 0,C 180,E1 -10194.117,E2 -10194.117} C_VEL
LIN {X 0,Y 419.238,Z 536.715,A -85,B 0,C 180,E1 -10196.641,E2 -10196.641} C_VEL
LIN {X 0,Y 418.314,Z 532.381,A -85,B 0,C 180,E1 -10197.678,E2 -10197.678} C_VEL
LIN {X 0,Y 418.236,Z 532.39,A -85,B 0,C 180,E1 -10201.018,E2 -10201.018} C_VEL
LIN {X 0,Y 418.245,Z 532.39,A -85,B 0,C 180,E1 -10203.675,E2 -10203.675} C_VEL
LIN {X 0,Y 418.243,Z 532.39,A -85,B 0,C 180,E1 -10207.222,E2 -10207.222} C_VEL
LIN {X 0,Y 418.261,Z 532.39,A -85,B 0,C 180,E1 -10209.679,E2 -10209.679} C_VEL
LIN {X 0,Y 418.242,Z 532.387,A -85,B 0,C 180,E1 -10212.322,E2 -10212.322} C_VEL
LIN {X 0,Y 418.232,Z 532.39,A -85,B 0,C 180,E1 -10215.108,E2 -10215.108} C_VEL
LIN {X 0,Y 418.249,Z 532.388,A -85,B 0,C 180,E1 -10217.767,E2 -10217.767} C_VEL
LIN {X 0,Y 418.261,Z 532.381,A -85,B 0,C 180,E1 -10220.615,E2 -10220.615} C_VEL
LIN {X 0,Y 418.239,Z 532.387,A -85,B 0,C 180,E1 -10223.975,E2 -10223.975} C_VEL
LIN {X 0,Y 418.249,Z 532.385,A -85,B 0,C 180,E1 -10227.155,E2 -10227.155} C_VEL
LIN {X 0,Y 418.266,Z 532.382,A -85,B 0,C 180,E1 -10230.838,E2 -10230.838} C_VEL
LIN {X 0,Y 418.261,Z 532.383,A -85,B 0,C 180,E1 -10234.095,E2 -10234.095} C_VEL
LIN {X 0,Y 418.228,Z 532.385,A -85,B 0,C 180,E1 -10237.263,E2 -10237.263} C_VEL
LIN {X 0,Y 418.273,Z 532.374,A -85,B 0,C 180,E1 -10240.363,E2 -10240.363} C_VEL
LIN {X 0,Y 418.306,Z 532.378,A -85,B 0,C 180,E1 -10243.404,E2 -10243.404} C_VEL
LIN {X 0,Y 418.344,Z 532.374,A -85,B 0,C 180,E1 -10246.993,E2 -10246.993} C_VEL
LIN {X 0,Y 418.349,Z 532.371,A -85,B 0,C 180,E1 -10250.328,E2 -10250.328} C_VEL
LIN {X 0,Y 418.483,Z 532.357,A -85,B 0,C 180,E1 -10253.248,E2 -10253.248} C_VEL
LIN {X 0,Y 418.332,Z 532.374,A -85,B 0,C 180,E1 -10255.181,E2 -10255.181} C_VEL
LIN {X 0,Y 418.534,Z 532.346,A -85,B 0,C 180,E1 -10258.075,E2 -10258.075} C_VEL
LIN {X 0,Y 418.663,Z 532.334,A -85,B 0,C 180,E1 -10260,E2 -10260} C_VEL
LIN {X 0,Y 418.502,Z 532.352,A -85,B 0,C 180,E1 -10262.887,E2 -10262.887} C_VEL
LIN {X 0,Y 418.482,Z 532.355,A -85,B 0,C 180,E1 -10266.641,E2 -10266.641} C_VEL
LIN {X 0,Y 418.388,Z 532.367,A -85,B 0,C 180,E1 -10268.695,E2 -10268.695} C_VEL
LIN {X 0,Y 418.324,Z 532.378,A -85,B 0,C 180,E1 -10271.63,E2 -10271.63} C_VEL
LIN {X 0,Y 418.295,Z 532.381,A -85,B 0,C 180,E1 -10274.597,E2 -10274.597} C_VEL
LIN {X 0,Y 418.275,Z 532.387,A -85,B 0,C 180,E1 -10277.604,E2 -10277.604} C_VEL
LIN {X 0,Y 418.237,Z 532.387,A -85,B 0,C 180,E1 -10280.663,E2 -10280.663} C_VEL
LIN {X 0,Y 418.275,Z 532.385,A -85,B 0,C 180,E1 -10283.781,E2 -10283.781} C_VEL
LIN {X 0,Y 418.317,Z 532.521,A -85,B 0,C 180,E1 -10286.235,E2 -10286.235} C_VEL
LIN {X 0,Y 420.394,Z 543.056,A -85,B 0,C 180,E1 -10289,E2 -10289} C_VEL
